LIN {X 0,Y 418.246,Z 332.012,A -85,B 0,C 180,E1 -10220.619,E2 -10220.619} C_VEL
LIN {X 0,Y 418.235,Z 332.015,A -85,B 0,C 180,E1 -10223.975,E2 -10223.975} C_VEL
LIN {X 0,Y 418.248,Z 332.008,A -85,B 0,C 180,E1 -10227.156,E2 -10227.156} C_VEL
LIN {X 0,Y 418.251,Z 331.996,A -85,B 0,C 180,E1 -10230.837,E2 -10230.837} C_VEL
LIN {X 0,Y 418.226,Z 332.013,A -85,B 0,C 180,E1 -10234.093,E2 -10234.093} C_VEL
LIN {X 0,Y 418.221,Z 332.012,A -85,B 0,C 180,E1 -10237.263,E2 -10237.263} C_VEL
LIN {X 0,Y 418.272,Z 332.006,A -85,B 0,C 180,E1 -10240.364,E2 -10240.364} C_VEL
LIN {X 0,Y 418.304,Z 332.002,A -85,B 0,C 180,E1 -10243.404,E2 -10243.404} C_VEL
LIN {X 0,Y 418.334,Z 331.998,A -85,B 0,C 180,E1 -10247,E2 -10247} C_VEL
LIN {X 0,Y 418.306,Z 332.002,A -85,B 0,C 180,E1 -10250.328,E2 -10250.328} C_VEL
LIN {X 0,Y 418.43,Z 331.983,A -85,B 0,C 180,E1 -10253.248,E2 -10253.248} C_VEL
LIN {X 0,Y 418.304,Z 332.004,A -85,B 0,C 180,E1 -10255.181,E2 -10255.181} C_VEL
LIN {X 0,Y 418.521,Z 331.97,A -85,B 0,C 180,E1 -10258.076,E2 -10258.076} C_VEL
LIN {X 0,Y 418.395,Z 331.993,A -85,B 0,C 180,E1 -10260.963,E2 -10260.963} C_VEL
LIN {X 0,Y 418.478,Z 331.976,A -85,B 0,C 180,E1 -10262.888,E2 -10262.888} C_VEL
LIN {X 0,Y 418.453,Z 331.982,A -85,B 0,C 180,E1 -10266.598,E2 -10266.598} C_VEL
LIN {X 0,Y 418.325,Z 332.001,A -85,B 0,C 180,E1 -10269.672,E2 -10269.672} C_VEL
LIN {X 0,Y 418.336,Z 331.996,A -85,B 0,C 180,E1 -10273.001,E2 -10273.001} C_VEL
LIN {X 0,Y 418.302,Z 332,A -85,B 0,C 180,E1 -10276.736,E2 -10276.736} C_VEL
LIN {X 0,Y 418.261,Z 332.005,A -85,B 0,C 180,E1 -10279.791,E2 -10279.791} C_VEL
LIN {X 0,Y 418.224,Z 332.016,A -85,B 0,C 180,E1 -10282.737,E2 -10282.737} C_VEL
LIN {X 0,Y 418.263,Z 332.006,A -85,B 0,C 180,E1 -10285.905,E2 -10285.905} C_VEL
LIN {X 0,Y 418.258,Z 332.01,A -85,B 0,C 180,E1 -10289.163,E2 -10289.163} C_VEL
LIN {X 0,Y 418.251,Z 332.012,A -85,B 0,C 180,E1 -10292.845,E2 -10292.845} C_VEL
LIN {X 0,Y 418.239,Z 332.012,A -85,B 0,C 180,E1 -10296.239,E2 -10296.239} C_VEL
LIN {X 0,Y 418.24,Z 332.008,A -85,B 0,C 180,E1 -10299.684,E2 -10299.684} C_VEL
LIN {X 0,Y 418.226,Z 332.014,A -85,B 0,C 180,E1 -10302.322,E2 -10302.322} C_VEL
LIN {X 0,Y 418.233,Z 332.013,A -85,B 0,C 180,E1 -10305.11,E2 -10305.11} C_VEL
LIN {X 0,Y 418.238,Z 332.013,A -85,B 0,C 180,E1 -10307.768,E2 -10307.768} C_VEL
LIN {X 0,Y 418.259,Z 332.011,A -85,B 0,C 180,E1 -10310.619,E2 -10310.619} C_VEL
LIN {X 0,Y 418.246,Z 332.014,A -85,B 0,C 180,E1 -10313.977,E2 -10313.977} C_VEL
LIN {X 0,Y 418.258,Z 332.108,A -85,B 0,C 180,E1 -10317.157,E2 -10317.157} C_VEL
LIN {X 0,Y 421.168,Z 344.799,A -85,B 0,C 180,E1 -10320.196,E2 -10320.196} C_VEL
LIN {X 0,Y 421.536,Z 346.615,A -85,B 0,C 180,E1 -10320.615,E2 -10320.615} C_VEL
LIN {X 0,Y 424.436,Z 354.758,A -85,B 0,C 180,E1 -10320.961,E2 -10320.961} C_VEL
LIN {X 0,Y 427.981,Z 370.411,A -85,B 0,C 180,E1 -10321.469,E2 -10321.469} C_VEL
LIN {X 0,Y 426.182,Z 483.541,A -85,B 0,C 180,E1 -10323.429,E2 -10323.429} C_VEL
LIN {X 0,Y 425.633,Z 498.284,A -85,B 0,C 180,E1 -10323.888,E2 -10323.888} C_VEL
LIN {X 0,Y 424.959,Z 512.346,A -85,B 0,C 180,E1 -10324.534,E2 -10324.534} C_VEL
LIN {X 0,Y 424.111,Z 524.49,A -85,B 0,C 180,E1 -10325.266,E2 -10325.266} C_VEL
LIN {X 0,Y 423.088,Z 537.105,A -85,B 0,C 180,E1 -10326.23,E2 -10326.23} C_VEL
LIN {X 0,Y 422.044,Z 548.902,A -85,B 0,C 180,E1 -10327.352,E2 -10327.352} C_VEL
LIN {X 0,Y 421.019,Z 559.619,A -85,B 0,C 180,E1 -10328.596,E2 -10328.596} C_VEL
LIN {X 0,Y 420.156,Z 569.213,A -85,B 0,C 180,E1 -10329.947,E2 -10329.947} C_VEL
LIN {X 0,Y 419.256,Z 577.982,A -85,B 0,C 180,E1 -10331.428,E2 -10331.428} C_VEL
LIN {X 0,Y 418.484,Z 586.467,A -85,B 0,C 180,E1 -10333.189,E2 -10333.189} C_VEL
LIN {X 0,Y 417.905,Z 593.022,A -85,B 0,C 180,E1 -10334.891,E2 -10334.891} C_VEL
LIN {X 0,Y 417.698,Z 595.505,A -85,B 0,C 180,E1 -10335.661,E2 -10335.661} C_VEL
LIN {X 0,Y 416.879,Z 597.766,A -85,B 0,C 180,E1 -10336.404,E2 -10336.404} C_VEL
LIN {X 0,Y 413.8,Z 601.016,A -85,B 0,C 180,E1 -10337.624,E2 -10337.624} C_VEL
LIN {X 0,Y 411.23,Z 603.194,A -85,B 0,C 180,E1 -10338.629,E2 -10338.629} C_VEL
LIN {X 0,Y 410.083,Z 604.573,A -85,B 0,C 180,E1 -10339.42,E2 -10339.42} C_VEL
LIN {X 0,Y 409.964,Z 604.953,A -85,B 0,C 180,E1 -10339.69,E2 -10339.69} C_VEL
LIN {X 0,Y 409.89,Z 606.657,A -85,B 0,C 180,E1 -10341.123,E2 -10341.123} C_VEL
LIN {X 0,Y 409.943,Z 607.798,A -85,B 0,C 180,E1 -10343.108,E2 -10343.108} C_VEL
LIN {X 0,Y 409.98,Z 607.87,A -85,B 0,C 180,E1 -10344.097,E2 -10344.097} C_VEL
LIN {X 0,Y 409.924,Z 607.031,A -85,B 0,C 180,E1 -10346.068,E2 -10346.068} C_VEL
LIN {X 0,Y 410.03,Z 604.86,A -85,B 0,C 180,E1 -10348.036,E2 -10348.036} C_VEL
LIN {X 0,Y 410.104,Z 601.318,A -85,B 0,C 180,E1 -10350,E2 -10350} C_VEL
LIN {X 0,Y 410.342,Z 596.299,A -85,B 0,C 180,E1 -10351.963,E2 -10351.963} C_VEL
LIN {X 0,Y 410.74,Z 591.435,A -85,B 0,C 180,E1 -10353.433,E2 -10353.433} C_VEL
LIN {X 0,Y 411.265,Z 584.464,A -85,B 0,C 180,E1 -10355.147,E2 -10355.147} C_VEL
LIN {X 0,Y 412.002,Z 577.174,A -85,B 0,C 180,E1 -10356.612,E2 -10356.612} C_VEL
LIN {X 0,Y 412.81,Z 568.431,A -85,B 0,C 180,E1 -10358.074,E2 -10358.074} C_VEL
LIN {X 0,Y 413.732,Z 557.988,A -85,B 0,C 180,E1 -10359.516,E2 -10359.516} C_VEL
LIN {X 0,Y 414.646,Z 547.174,A -85,B 0,C 180,E1 -10360.745,E2 -10360.745} C_VEL
LIN {X 0,Y 415.586,Z 535.499,A -85,B 0,C 180,E1 -10361.832,E2 -10361.832} C_VEL
LIN {X 0,Y 416.513,Z 522.632,A -85,B 0,C 180,E1 -10362.795,E2 -10362.795} C_VEL
LIN {X 0,Y 417.36,Z 509.181,A -85,B 0,C 180,E1 -10363.573,E2 -10363.573} C_VEL
LIN {X 0,Y 417.958,Z 495.939,A -85,B 0,C 180,E1 -10364.143,E2 -10364.143} C_VEL
LIN {X 0,Y 418.392,Z 481.346,A -85,B 0,C 180,E1 -10364.562,E2 -10364.562} C_VEL
LIN {X 0,Y 419.816,Z 370.702,A -85,B 0,C 180,E1 -10366.485,E2 -10366.485} C_VEL
LIN {X 0,Y 415.593,Z 351.069,A -85,B 0,C 180,E1 -10367.062,E2 -10367.062} C_VEL
LIN {X 0,Y 414.048,Z 346.577,A -85,B 0,C 180,E1 -10367.248,E2 -10367.248} C_VEL
LIN {X 0,Y 411.854,Z 335.866,A -85,B 0,C 180,E1 -10369.695,E2 -10369.695} C_VEL
LIN {X 0,Y 411.239,Z 332.889,A -85,B 0,C 180,E1 -10370.435,E2 -10370.435} C_VEL
LIN {X 0,Y 411.228,Z 332.887,A -85,B 0,C 180,E1 -10374.215,E2 -10374.215} C_VEL
LIN {X 0,Y 411.261,Z 332.883,A -85,B 0,C 180,E1 -10377.477,E2 -10377.477} C_VEL
LIN {X 0,Y 411.19,Z 332.888,A -85,B 0,C 180,E1 -10380.847,E2 -10380.847} C_VEL
LIN {X 0,Y 411.206,Z 332.885,A -85,B 0,C 180,E1 -10384.332,E2 -10384.332} C_VEL
LIN {X 0,Y 411.199,Z 332.889,A -85,B 0,C 180,E1 -10387.972,E2 -10387.972} C_VEL
LIN {X 0,Y 411.18,Z 332.876,A -85,B 0,C 180,E1 -10390.503,E2 -10390.503} C_VEL
LIN {X 0,Y 411.171,Z 332.892,A -85,B 0,C 180,E1 -10393.132,E2 -10393.132} C_VEL
LIN {X 0,Y 411.164,Z 332.893,A -85,B 0,C 180,E1 -10395.88,E2 -10395.88} C_VEL
LIN {X 0,Y 411.159,Z 332.888,A -85,B 0,C 180,E1 -10398.771,E2 -10398.771} C_VEL
LIN {X 0,Y 411.186,Z 332.883,A -85,B 0,C 180,E1 -10402.025,E2 -10402.025} C_VEL
LIN {X 0,Y 411.198,Z 332.885,A -85,B 0,C 180,E1 -10405.665,E2 -10405.665} C_VEL
LIN {X 0,Y 411.182,Z 332.895,A -85,B 0,C 180,E1 -10409.151,E2 -10409.151} C_VEL
LIN {X 0,Y 411.251,Z 332.872,A -85,B 0,C 180,E1 -10412.521,E2 -10412.521} C_VEL
LIN {X 0,Y 411.202,Z 332.886,A -85,B 0,C 180,E1 -10415.783,E2 -10415.783} C_VEL
LIN {X 0,Y 411.186,Z 332.88,A -85,B 0,C 180,E1 -10418.965,E2 -10418.965} C_VEL
LIN {X 0,Y 411.235,Z 332.879,A -85,B 0,C 180,E1 -10422.084,E2 -10422.084} C_VEL
LIN {X 0,Y 411.247,Z 332.878,A -85,B 0,C 180,E1 -10425.146,E2 -10425.146} C_VEL
LIN {X 0,Y 411.27,Z 332.866,A -85,B 0,C 180,E1 -10428.166,E2 -10428.166} C_VEL
LIN {X 0,Y 411.427,Z 332.859,A -85,B 0,C 180,E1 -10432.191,E2 -10432.191} C_VEL
LIN {X 0,Y 411.432,Z 332.853,A -85,B 0,C 180,E1 -10434.117,E2 -10434.117} C_VEL
LIN {X 0,Y 411.493,Z 332.847,A -85,B 0,C 180,E1 -10438.042,E2 -10438.042} C_VEL
LIN {X 0,Y 411.487,Z 332.848,A -85,B 0,C 180,E1 -10441.957,E2 -10441.957} C_VEL
LIN {X 0,Y 411.405,Z 332.861,A -85,B 0,C 180,E1 -10445.883,E2 -10445.883} C_VEL
LIN {X 0,Y 411.298,Z 332.867,A -85,B 0,C 180,E1 -10448.846,E2 -10448.846} C_VEL
LIN {X 0,Y 411.269,Z 332.878,A -85,B 0,C 180,E1 -10451.833,E2 -10451.833} C_VEL
LIN {X 0,Y 411.247,Z 332.875,A -85,B 0,C 180,E1 -10454.853,E2 -10454.853} C_VEL
LIN {X 0,Y 411.233,Z 332.883,A -85,B 0,C 180,E1 -10457.916,E2 -10457.916} C_VEL
LIN {X 0,Y 411.185,Z 332.879,A -85,B 0,C 180,E1 -10461.034,E2 -10461.034} C_VEL
LIN {X 0,Y 411.201,Z 332.888,A -85,B 0,C 180,E1 -10464.217,E2 -10464.217} C_VEL
LIN {X 0,Y 411.179,Z 332.887,A -85,B 0,C 180,E1 -10467.483,E2 -10467.483} C_VEL
LIN {X 0,Y 411.179,Z 332.886,A -85,B 0,C 180,E1 -10470.848,E2 -10470.848} C_VEL
LIN {X 0,Y 411.197,Z 332.888,A -85,B 0,C 180,E1 -10474.334,E2 -10474.334} C_VEL
LIN {X 0,Y 411.188,Z 332.892,A -85,B 0,C 180,E1 -10477.974,E2 -10477.974} C_VEL
LIN {X 0,Y 411.175,Z 332.884,A -85,B 0,C 180,E1 -10480.505,E2 -10480.505} C_VEL
LIN {X 0,Y 411.167,Z 332.889,A -85,B 0,C 180,E1 -10483.134,E2 -10483.134} C_VEL
LIN {X 0,Y 411.162,Z 332.896,A -85,B 0,C 180,E1 -10485.882,E2 -10485.882} C_VEL
LIN {X 0,Y 411.157,Z 332.893,A -85,B 0,C 180,E1 -10488.773,E2 -10488.773} C_VEL
LIN {X 0,Y 411.187,Z 332.895,A -85,B 0,C 180,E1 -10492.027,E2 -10492.027} C_VEL
LIN {X 0,Y 411.203,Z 332.894,A -85,B 0,C 180,E1 -10495.667,E2 -10495.667} C_VEL
LIN {X 0,Y 411.188,Z 332.893,A -85,B 0,C 180,E1 -10499.153,E2 -10499.153} C_VEL
LIN {X 0,Y 411.232,Z 332.987,A -85,B 0,C 180,E1 -10500.044,E2 -10500.044} C_VEL
LIN {X 0,Y 414.112,Z 345.944,A -85,B 0,C 180,E1 -10502.728,E2 -10502.728} C_VEL
LIN {X 0,Y 415.486,Z 353.214,A -85,B 0,C 180,E1 -10504.18,E2 -10504.18} C_VEL
LIN {X 0,Y 414.529,Z 367.772,A -85,B 0,C 180,E1 -10506.824,E2 -10506.824} C_VEL
LIN {X 0,Y 419.611,Z 397.438,A -85,B 0,C 180,E1 -10507.622,E2 -10507.622} C_VEL
LIN {X 0,Y 418.121,Z 505.146,A -85,B 0,C 180,E1 -10509.492,E2 -10509.492} C_VEL
LIN {X 0,Y 417.563,Z 519.304,A -85,B 0,C 180,E1 -10509.913,E2 -10509.913} C_VEL
LIN {X 0,Y 416.82,Z 532.559,A -85,B 0,C 180,E1 -10510.49,E2 -10510.49} C_VEL
LIN {X 0,Y 416.007,Z 545.949,A -85,B 0,C 180,E1 -10511.278,E2 -10511.278} C_VEL
LIN {X 0,Y 415.023,Z 558.885,A -85,B 0,C 180,E1 -10512.254,E2 -10512.254} C_VEL
LIN {X 0,Y 413.918,Z 570.625,A -85,B 0,C 180,E1 -10513.351,E2 -10513.351} C_VEL
LIN {X 0,Y 413.086,Z 580.397,A -85,B 0,C 180,E1 -10514.458,E2 -10514.458} C_VEL
LIN {X 0,Y 412.209,Z 591.218,A -85,B 0,C 180,E1 -10515.939,E2 -10515.939} C_VEL
LIN {X 0,Y 411.522,Z 600.144,A -85,B 0,C 180,E1 -10517.424,E2 -10517.424} C_VEL
LIN {X 0,Y 410.96,Z 607.561,A -85,B 0,C 180,E1 -10518.908,E2 -10518.908} C_VEL
LIN {X 0,Y 410.45,Z 614.649,A -85,B 0,C 180,E1 -10520.639,E2 -10520.639} C_VEL
LIN {X 0,Y 410.157,Z 621.011,A -85,B 0,C 180,E1 -10522.617,E2 -10522.617} C_VEL
LIN {X 0,Y 410.034,Z 624.648,A -85,B 0,C 180,E1 -10524.097,E2 -10524.097} C_VEL
LIN {X 0,Y 409.92,Z 628.205,A -85,B 0,C 180,E1 -10526.068,E2 -10526.068} C_VEL
LIN {X 0,Y 409.964,Z 630.356,A -85,B 0,C 180,E1 -10528.035,E2 -10528.035} C_VEL
LIN {X 0,Y 409.924,Z 631.15,A -85,B 0,C 180,E1 -10530,E2 -10530} C_VEL
LIN {X 0,Y 409.964,Z 630.613,A -85,B 0,C 180,E1 -10531.965,E2 -10531.965} C_VEL
LIN {X 0,Y 409.919,Z 628.737,A -85,B 0,C 180,E1 -10533.932,E2 -10533.932} C_VEL
LIN {X 0,Y 410.034,Z 625.471,A -85,B 0,C 180,E1 -10535.903,E2 -10535.903} C_VEL
LIN {X 0,Y 410.161,Z 622.032,A -85,B 0,C 180,E1 -10537.383,E2 -10537.383} C_VEL
LIN {X 0,Y 410.51,Z 616.109,A -85,B 0,C 180,E1 -10539.36,E2 -10539.36} C_VEL
LIN {X 0,Y 411.005,Z 609.456,A -85,B 0,C 180,E1 -10541.091,E2 -10541.091} C_VEL
LIN {X 0,Y 411.737,Z 601.197,A -85,B 0,C 180,E1 -10542.82,E2 -10542.82} C_VEL
LIN {X 0,Y 412.532,Z 592.598,A -85,B 0,C 180,E1 -10544.301,E2 -10544.301} C_VEL
LIN {X 0,Y 413.546,Z 582.197,A -85,B 0,C 180,E1 -10545.778,E2 -10545.778} C_VEL
LIN {X 0,Y 414.765,Z 570.585,A -85,B 0,C 180,E1 -10547.122,E2 -10547.122} C_VEL
LIN {X 0,Y 415.872,Z 559.001,A -85,B 0,C 180,E1 -10548.218,E2 -10548.218} C_VEL
LIN {X 0,Y 416.962,Z 546.906,A -85,B 0,C 180,E1 -10549.142,E2 -10549.142} C_VEL
LIN {X 0,Y 417.909,Z 533.112,A -85,B 0,C 180,E1 -10549.974,E2 -10549.974} C_VEL
LIN {X 0,Y 418.786,Z 519.614,A -85,B 0,C 180,E1 -10550.571,E2 -10550.571} C_VEL
LIN {X 0,Y 419.409,Z 505.937,A -85,B 0,C 180,E1 -10550.988,E2 -10550.988} C_VEL
LIN {X 0,Y 421.196,Z 399.896,A -85,B 0,C 180,E1 -10552.852,E2 -10552.852} C_VEL
LIN {X 0,Y 420.511,Z 393.745,A -85,B 0,C 180,E1 -10553.008,E2 -10553.008} C_VEL
LIN {X 0,Y 415.325,Z 367.391,A -85,B 0,C 180,E1 -10553.851,E2 -10553.851} C_VEL
LIN {X 0,Y 416.283,Z 355.716,A -85,B 0,C 180,E1 -10556.036,E2 -10556.036} C_VEL
LIN {X 0,Y 414.111,Z 344.618,A -85,B 0,C 180,E1 -10558.371,E2 -10558.371} C_VEL
LIN {X 0,Y 411.208,Z 332.891,A -85,B 0,C 180,E1 -10561.008,E2 -10561.008} C_VEL
LIN {X 0,Y 411.202,Z 332.891,A -85,B 0,C 180,E1 -10564.333,E2 -10564.333} C_VEL
LIN {X 0,Y 411.19,Z 332.882,A -85,B 0,C 180,E1 -10567.973,E2 -10567.973} C_VEL
LIN {X 0,Y 411.158,Z 332.886,A -85,B 0,C 180,E1 -10571.227,E2 -10571.227} C_VEL
LIN {X 0,Y 411.169,Z 332.889,A -85,B 0,C 180,E1 -10574.49,E2 -10574.49} C_VEL
LIN {X 0,Y 411.17,Z 332.893,A -85,B 0,C 180,E1 -10578.194,E2 -10578.194} C_VEL
LIN {X 0,Y 411.21,Z 332.887,A -85,B 0,C 180,E1 -10580.775,E2 -10580.775} C_VEL
LIN {X 0,Y 411.19,Z 332.888,A -85,B 0,C 180,E1 -10584.471,E2 -10584.471} C_VEL
LIN {X 0,Y 411.199,Z 332.887,A -85,B 0,C 180,E1 -10586.873,E2 -10586.873} C_VEL
LIN {X 0,Y 411.203,Z 332.872,A -85,B 0,C 180,E1 -10590.649,E2 -10590.649} C_VEL
LIN {X 0,Y 411.185,Z 332.891,A -85,B 0,C 180,E1 -10593.616,E2 -10593.616} C_VEL
LIN {X 0,Y 411.185,Z 332.888,A -85,B 0,C 180,E1 -10596.852,E2 -10596.852} C_VEL
LIN {X 0,Y 411.203,Z 332.887,A -85,B 0,C 180,E1 -10600.051,E2 -10600.051} C_VEL
LIN {X 0,Y 411.252,Z 332.88,A -85,B 0,C 180,E1 -10603.131,E2 -10603.131} C_VEL
LIN {X 0,Y 411.293,Z 332.875,A -85,B 0,C 180,E1 -10606.897,E2 -10606.897} C_VEL
LIN {X 0,Y 411.26,Z 332.88,A -85,B 0,C 180,E1 -10610.161,E2 -10610.161} C_VEL
LIN {X 0,Y 411.379,Z 332.861,A -85,B 0,C 180,E1 -10613.132,E2 -10613.132} C_VEL
LIN {X 0,Y 411.276,Z 332.879,A -85,B 0,C 180,E1 -10615.099,E2 -10615.099} C_VEL
LIN {X 0,Y 411.49,Z 332.846,A -85,B 0,C 180,E1 -10618.043,E2 -10618.043} C_VEL
LIN {X 0,Y 411.497,Z 332.845,A -85,B 0,C 180,E1 -10621.958,E2 -10621.958} C_VEL
LIN {X 0,Y 411.412,Z 332.859,A -85,B 0,C 180,E1 -10626.6,E2 -10626.6} C_VEL
LIN {X 0,Y 411.307,Z 332.872,A -85,B 0,C 180,E1 -10628.847,E2 -10628.847} C_VEL
LIN {X 0,Y 411.27,Z 332.871,A -85,B 0,C 180,E1 -10631.834,E2 -10631.834} C_VEL
LIN {X 0,Y 411.247,Z 332.885,A -85,B 0,C 180,E1 -10634.854,E2 -10634.854} C_VEL
LIN {X 0,Y 411.236,Z 332.882,A -85,B 0,C 180,E1 -10637.916,E2 -10637.916} C_VEL
LIN {X 0,Y 411.187,Z 332.888,A -85,B 0,C 180,E1 -10641.035,E2 -10641.035} C_VEL
LIN {X 0,Y 411.212,Z 332.884,A -85,B 0,C 180,E1 -10644.217,E2 -10644.217} C_VEL
LIN {X 0,Y 411.252,Z 332.878,A -85,B 0,C 180,E1 -10647.479,E2 -10647.479} C_VEL
LIN {X 0,Y 411.183,Z 332.889,A -85,B 0,C 180,E1 -10650.849,E2 -10650.849} C_VEL
LIN {X 0,Y 411.2,Z 332.887,A -85,B 0,C 180,E1 -10654.335,E2 -10654.335} C_VEL
LIN {X 0,Y 411.186,Z 332.886,A -85,B 0,C 180,E1 -10657.975,E2 -10657.975} C_VEL
LIN {X 0,Y 411.159,Z 332.893,A -85,B 0,C 180,E1 -10661.229,E2 -10661.229} C_VEL
LIN {X 0,Y 411.173,Z 332.893,A -85,B 0,C 180,E1 -10664.492,E2 -10664.492} C_VEL
LIN {X 0,Y 411.175,Z 332.895,A -85,B 0,C 180,E1 -10668.196,E2 -10668.196} C_VEL
LIN {X 0,Y 411.223,Z 332.888,A -85,B 0,C 180,E1 -10670.778,E2 -10670.778} C_VEL
LIN {X 0,Y 411.199,Z 332.887,A -85,B 0,C 180,E1 -10674.473,E2 -10674.473} C_VEL
LIN {X 0,Y 411.227,Z 333.001,A -85,B 0,C 180,E1 -10676.774,E2 -10676.774} C_VEL
LIN {X 0,Y 414.352,Z 346.613,A -85,B 0,C 180,E1 -10680.095,E2 -10680.095} C_VEL
LIN {X 0,Y 414.484,Z 347.202,A -85,B 0,C 180,E1 -10680.167,E2 -10680.167} C_VEL
LIN {X 0,Y 418.19,Z 356.786,A -85,B 0,C 180,E1 -10680.595,E2 -10680.595} C_VEL
LIN {X 0,Y 421.558,Z 371.616,A -85,B 0,C 180,E1 -10681.088,E2 -10681.088} C_VEL
LIN {X 0,Y 419.636,Z 483.745,A -85,B 0,C 180,E1 -10683.058,E2 -10683.058} C_VEL
LIN {X 0,Y 419.091,Z 498.27,A -85,B 0,C 180,E1 -10683.516,E2 -10683.516} C_VEL
LIN {X 0,Y 418.362,Z 512.383,A -85,B 0,C 180,E1 -10684.17,E2 -10684.17} C_VEL
LIN {X 0,Y 417.409,Z 525.458,A -85,B 0,C 180,E1 -10684.974,E2 -10684.974} C_VEL
LIN {X 0,Y 416.369,Z 537.689,A -85,B 0,C 180,E1 -10685.933,E2 -10685.933} C_VEL
LIN {X 0,Y 415.361,Z 548.417,A -85,B 0,C 180,E1 -10686.967,E2 -10686.967} C_VEL
LIN {X 0,Y 414.346,Z 558.16,A -85,B 0,C 180,E1 -10688.09,E2 -10688.09} C_VEL
LIN {X 0,Y 413.431,Z 568.078,A -85,B 0,C 180,E1 -10689.47,E2 -10689.47} C_VEL
LIN {X 0,Y 412.376,Z 577.785,A -85,B 0,C 180,E1 -10691.107,E2 -10691.107} C_VEL
LIN {X 0,Y 411.689,Z 585.113,A -85,B 0,C 180,E1 -10692.619,E2 -10692.619} C_VEL
LIN {X 0,Y 411.096,Z 591.175,A -85,B 0,C 180,E1 -10694.126,E2 -10694.126} C_VEL
LIN {X 0,Y 410.647,Z 596.17,A -85,B 0,C 180,E1 -10695.632,E2 -10695.632} C_VEL
LIN {X 0,Y 410.302,Z 601.035,A -85,B 0,C 180,E1 -10697.516,E2 -10697.516} C_VEL
LIN {X 0,Y 410.06,Z 604.154,A -85,B 0,C 180,E1 -10699.133,E2 -10699.133} C_VEL
LIN {X 0,Y 409.964,Z 604.953,A -85,B 0,C 180,E1 -10699.69,E2 -10699.69} C_VEL
LIN {X 0,Y 409.241,Z 606.048,A -85,B 0,C 180,E1 -10700.496,E2 -10700.496} C_VEL
LIN {X 0,Y 406.418,Z 607.421,A -85,B 0,C 180,E1 -10701.816,E2 -10701.816} C_VEL
LIN {X 0,Y 404.05,Z 608.026,A -85,B 0,C 180,E1 -10702.889,E2 -10702.889} C_VEL
LIN {X 0,Y 403.004,Z 608.126,A -85,B 0,C 180,E1 -10703.719,E2 -10703.719} C_VEL
LIN {X 0,Y 402.901,Z 608.082,A -85,B 0,C 180,E1 -10704,E2 -10704} C_VEL
LIN {X 0,Y 402.84,Z 607.29,A -85,B 0,C 180,E1 -10705.998,E2 -10705.998} C_VEL
LIN {X 0,Y 402.957,Z 605.165,A -85,B 0,C 180,E1 -10708.001,E2 -10708.001} C_VEL
LIN {X 0,Y 403.019,Z 601.673,A -85,B 0,C 180,E1 -10710,E2 -10710} C_VEL
LIN {X 0,Y 403.262,Z 596.705,A -85,B 0,C 180,E1 -10711.997,E2 -10711.997} C_VEL
LIN {X 0,Y 403.752,Z 590.109,A -85,B 0,C 180,E1 -10713.992,E2 -10713.992} C_VEL
LIN {X 0,Y 404.512,Z 582.752,A -85,B 0,C 180,E1 -10715.733,E2 -10715.733} C_VEL
LIN {X 0,Y 405.267,Z 575.079,A -85,B 0,C 180,E1 -10717.223,E2 -10717.223} C_VEL
LIN {X 0,Y 406.132,Z 565.865,A -85,B 0,C 180,E1 -10718.709,E2 -10718.709} C_VEL
LIN {X 0,Y 407.011,Z 555.701,A -85,B 0,C 180,E1 -10720.067,E2 -10720.067} C_VEL
LIN {X 0,Y 408.003,Z 544.479,A -85,B 0,C 180,E1 -10721.299,E2 -10721.299} C_VEL
LIN {X 0,Y 409.005,Z 532.093,A -85,B 0,C 180,E1 -10722.403,E2 -10722.403} C_VEL
LIN {X 0,Y 409.894,Z 520.134,A -85,B 0,C 180,E1 -10723.257,E2 -10723.257} C_VEL
LIN {X 0,Y 410.686,Z 507.015,A -85,B 0,C 180,E1 -10723.988,E2 -10723.988} C_VEL
LIN {X 0,Y 411.368,Z 493.66,A -85,B 0,C 180,E1 -10724.532,E2 -10724.532} C_VEL
LIN {X 0,Y 411.735,Z 478.975,A -85,B 0,C 180,E1 -10724.93,E2 -10724.93} C_VEL
LIN {X 0,Y 413.261,Z 372.068,A -85,B 0,C 180,E1 -10726.804,E2 -10726.804} C_VEL
LIN {X 0,Y 409.161,Z 353.235,A -85,B 0,C 180,E1 -10727.372,E2 -10727.372} C_VEL
LIN {X 0,Y 406.897,Z 346.78,A -85,B 0,C 180,E1 -10727.641,E2 -10727.641} C_VEL
LIN {X 0,Y 404.186,Z 333.781,A -85,B 0,C 180,E1 -10730.682,E2 -10730.682} C_VEL
LIN {X 0,Y 404.171,Z 333.767,A -85,B 0,C 180,E1 -10733.574,E2 -10733.574} C_VEL
LIN {X 0,Y 404.185,Z 333.766,A -85,B 0,C 180,E1 -10735.765,E2 -10735.765} C_VEL
LIN {X 0,Y 404.197,Z 333.76,A -85,B 0,C 180,E1 -10737.999,E2 -10737.999} C_VEL
LIN {X 0,Y 404.14,Z 333.77,A -85,B 0,C 180,E1 -10741.557,E2 -10741.557} C_VEL
LIN {X 0,Y 404.185,Z 333.76,A -85,B 0,C 180,E1 -10745.015,E2 -10745.015} C_VEL
LIN {X 0,Y 404.157,Z 333.764,A -85,B 0,C 180,E1 -10748.755,E2 -10748.755} C_VEL
LIN {X 0,Y 404.121,Z 333.765,A -85,B 0,C 180,E1 -10751.598,E2 -10751.598} C_VEL
LIN {X 0,Y 404.142,Z 333.763,A -85,B 0,C 180,E1 -10754.521,E2 -10754.521} C_VEL
LIN {X 0,Y 404.132,Z 333.771,A -85,B 0,C 180,E1 -10757.294,E2 -10757.294} C_VEL
LIN {X 0,Y 404.165,Z 333.764,A -85,B 0,C 180,E1 -10759.954,E2 -10759.954} C_VEL
LIN {X 0,Y 404.13,Z 333.767,A -85,B 0,C 180,E1 -10763.124,E2 -10763.124} C_VEL
LIN {X 0,Y 404.138,Z 333.762,A -85,B 0,C 180,E1 -10766.186,E2 -10766.186} C_VEL
LIN {X 0,Y 404.138,Z 333.766,A -85,B 0,C 180,E1 -10769.714,E2 -10769.714} C_VEL
LIN {X 0,Y 404.185,Z 333.754,A -85,B 0,C 180,E1 -10773.122,E2 -10773.122} C_VEL
LIN {X 0,Y 404.151,Z 333.765,A -85,B 0,C 180,E1 -10776.424,E2 -10776.424} C_VEL
LIN {X 0,Y 404.182,Z 333.747,A -85,B 0,C 180,E1 -10779.873,E2 -10779.873} C_VEL
LIN {X 0,Y 404.206,Z 333.763,A -85,B 0,C 180,E1 -10782.992,E2 -10782.992} C_VEL
LIN {X 0,Y 404.273,Z 333.738,A -85,B 0,C 180,E1 -10786.938,E2 -10786.938} C_VEL
LIN {X 0,Y 404.243,Z 333.75,A -85,B 0,C 180,E1 -10789.988,E2 -10789.988} C_VEL
LIN {X 0,Y 404.371,Z 333.735,A -85,B 0,C 180,E1 -10793.012,E2 -10793.012} C_VEL
LIN {X 0,Y 404.257,Z 333.737,A -85,B 0,C 180,E1 -10795.013,E2 -10795.013} C_VEL
LIN {X 0,Y 404.462,Z 333.722,A -85,B 0,C 180,E1 -10798.008,E2 -10798.008} C_VEL
LIN {X 0,Y 404.456,Z 333.724,A -85,B 0,C 180,E1 -10801.991,E2 -10801.991} C_VEL
LIN {X 0,Y 404.355,Z 333.74,A -85,B 0,C 180,E1 -10805.986,E2 -10805.986} C_VEL
LIN {X 0,Y 404.247,Z 333.744,A -85,B 0,C 180,E1 -10809.002,E2 -10809.002} C_VEL
LIN {X 0,Y 404.242,Z 333.755,A -85,B 0,C 180,E1 -10812.042,E2 -10812.042} C_VEL
LIN {X 0,Y 404.193,Z 333.752,A -85,B 0,C 180,E1 -10815.118,E2 -10815.118} C_VEL
LIN {X 0,Y 404.192,Z 333.764,A -85,B 0,C 180,E1 -10818.239,E2 -10818.239} C_VEL
LIN {X 0,Y 404.127,Z 333.758,A -85,B 0,C 180,E1 -10821.42,E2 -10821.42} C_VEL
LIN {X 0,Y 404.154,Z 333.762,A -85,B 0,C 180,E1 -10824.667,E2 -10824.667} C_VEL
LIN {X 0,Y 404.12,Z 333.772,A -85,B 0,C 180,E1 -10828.005,E2 -10828.005} C_VEL
LIN {X 0,Y 404.135,Z 333.765,A -85,B 0,C 180,E1 -10830.286,E2 -10830.286} C_VEL
LIN {X 0,Y 404.136,Z 333.768,A -85,B 0,C 180,E1 -10833.813,E2 -10833.813} C_VEL
LIN {X 0,Y 404.128,Z 333.766,A -85,B 0,C 180,E1 -10836.876,E2 -10836.876} C_VEL
LIN {X 0,Y 404.14,Z 333.764,A -85,B 0,C 180,E1 -10840.081,E2 -10840.081} C_VEL
LIN {X 0,Y 404.146,Z 333.764,A -85,B 0,C 180,E1 -10843.084,E2 -10843.084} C_VEL
LIN {X 0,Y 404.142,Z 333.77,A -85,B 0,C 180,E1 -10845.927,E2 -10845.927} C_VEL
LIN {X 0,Y 404.112,Z 333.77,A -85,B 0,C 180,E1 -10848.636,E2 -10848.636} C_VEL
LIN {X 0,Y 404.145,Z 333.773,A -85,B 0,C 180,E1 -10851.494,E2 -10851.494} C_VEL
LIN {X 0,Y 404.181,Z 333.768,A -85,B 0,C 180,E1 -10854.985,E2 -10854.985} C_VEL
LIN {X 0,Y 404.139,Z 333.77,A -85,B 0,C 180,E1 -10858.555,E2 -10858.555} C_VEL
LIN {X 0,Y 404.17,Z 333.819,A -85,B 0,C 180,E1 -10859.718,E2 -10859.718} C_VEL
LIN {X 0,Y 407.113,Z 346.963,A -85,B 0,C 180,E1 -10862.498,E2 -10862.498} C_VEL
LIN {X 0,Y 408.573,Z 354.383,A -85,B 0,C 180,E1 -10864.012,E2 -10864.012} C_VEL
LIN {X 0,Y 407.668,Z 367.447,A -85,B 0,C 180,E1 -10866.444,E2 -10866.444} C_VEL
LIN {X 0,Y 412.999,Z 398.828,A -85,B 0,C 180,E1 -10867.309,E2 -10867.309} C_VEL
LIN {X 0,Y 411.419,Z 504.838,A -85,B 0,C 180,E1 -10869.175,E2 -10869.175} C_VEL
LIN {X 0,Y 410.813,Z 519.039,A -85,B 0,C 180,E1 -10869.601,E2 -10869.601} C_VEL
LIN {X 0,Y 410.008,Z 533.257,A -85,B 0,C 180,E1 -10870.239,E2 -10870.239} C_VEL
LIN {X 0,Y 409.086,Z 547.047,A -85,B 0,C 180,E1 -10871.079,E2 -10871.079} C_VEL
LIN {X 0,Y 408.083,Z 559.737,A -85,B 0,C 180,E1 -10872.071,E2 -10872.071} C_VEL
LIN {X 0,Y 406.952,Z 571.293,A -85,B 0,C 180,E1 -10873.186,E2 -10873.186} C_VEL
LIN {X 0,Y 405.999,Z 581.904,A -85,B 0,C 180,E1 -10874.437,E2 -10874.437} C_VEL
LIN {X 0,Y 405.116,Z 592.444,A -85,B 0,C 180,E1 -10875.944,E2 -10875.944} C_VEL
LIN {X 0,Y 404.403,Z 601.131,A -85,B 0,C 180,E1 -10877.454,E2 -10877.454} C_VEL
LIN {X 0,Y 403.724,Z 609.438,A -85,B 0,C 180,E1 -10879.215,E2 -10879.215} C_VEL
LIN {X 0,Y 403.289,Z 616.111,A -85,B 0,C 180,E1 -10880.977,E2 -10880.977} C_VEL
LIN {X 0,Y 403.067,Z 622.03,A -85,B 0,C 180,E1 -10882.99,E2 -10882.99} C_VEL
LIN {X 0,Y 402.903,Z 626.352,A -85,B 0,C 180,E1 -10884.997,E2 -10884.997} C_VEL
LIN {X 0,Y 402.822,Z 629.215,A -85,B 0,C 180,E1 -10887,E2 -10887} C_VEL
LIN {X 0,Y 402.86,Z 630.705,A -85,B 0,C 180,E1 -10889,E2 -10889} C_VEL
LIN {X 0,Y 402.86,Z 630.851,A -85,B 0,C 180,E1 -10891,E2 -10891} C_VEL
LIN {X 0,Y 402.818,Z 629.666,A -85,B 0,C 180,E1 -10893,E2 -10893} C_VEL
LIN {X 0,Y 402.903,Z 627.132,A -85,B 0,C 180,E1 -10895.003,E2 -10895.003} C_VEL
LIN {X 0,Y 403.067,Z 623.159,A -85,B 0,C 180,E1 -10897.01,E2 -10897.01} C_VEL
LIN {X 0,Y 403.345,Z 617.63,A -85,B 0,C 180,E1 -10899.022,E2 -10899.022} C_VEL
LIN {X 0,Y 403.791,Z 611.405,A -85,B 0,C 180,E1 -10900.784,E2 -10900.784} C_VEL
LIN {X 0,Y 404.621,Z 603.664,A -85,B 0,C 180,E1 -10902.539,E2 -10902.539} C_VEL
LIN {X 0,Y 405.317,Z 595.603,A -85,B 0,C 180,E1 -10904.049,E2 -10904.049} C_VEL
LIN {X 0,Y 406.341,Z 585.907,A -85,B 0,C 180,E1 -10905.55,E2 -10905.55} C_VEL
LIN {X 0,Y 407.496,Z 575.166,A -85,B 0,C 180,E1 -10906.92,E2 -10906.92} C_VEL
LIN {X 0,Y 408.782,Z 563.292,A -85,B 0,C 180,E1 -10908.156,E2 -10908.156} C_VEL
LIN {X 0,Y 409.881,Z 551.787,A -85,B 0,C 180,E1 -10909.131,E2 -10909.131} C_VEL
LIN {X 0,Y 410.919,Z 538.966,A -85,B 0,C 180,E1 -10910.002,E2 -10910.002} C_VEL
LIN {X 0,Y 411.766,Z 526.096,A -85,B 0,C 180,E1 -10910.676,E2 -10910.676} C_VEL
LIN {X 0,Y 412.659,Z 511.492,A -85,B 0,C 180,E1 -10911.217,E2 -10911.217} C_VEL
LIN {X 0,Y 413.077,Z 496.943,A -85,B 0,C 180,E1 -10911.554,E2 -10911.554} C_VEL
LIN {X 0,Y 414.759,Z 399.127,A -85,B 0,C 180,E1 -10913.275,E2 -10913.275} C_VEL
LIN {X 0,Y 411.006,Z 378.832,A -85,B 0,C 180,E1 -10913.906,E2 -10913.906} C_VEL
LIN {X 0,Y 408.598,Z 367.199,A -85,B 0,C 180,E1 -10914.306,E2 -10914.306} C_VEL
LIN {X 0,Y 409.418,Z 357.116,A -85,B 0,C 180,E1 -10916.232,E2 -10916.232} C_VEL
LIN {X 0,Y 407.275,Z 346.336,A -85,B 0,C 180,E1 -10918.548,E2 -10918.548} C_VEL
LIN {X 0,Y 404.139,Z 333.771,A -85,B 0,C 180,E1 -10921.445,E2 -10921.445} C_VEL
LIN {X 0,Y 404.181,Z 333.763,A -85,B 0,C 180,E1 -10925.015,E2 -10925.015} C_VEL
LIN {X 0,Y 404.149,Z 333.764,A -85,B 0,C 180,E1 -10928.756,E2 -10928.756} C_VEL
LIN {X 0,Y 404.117,Z 333.763,A -85,B 0,C 180,E1 -10931.599,E2 -10931.599} C_VEL
LIN {X 0,Y 404.139,Z 333.764,A -85,B 0,C 180,E1 -10934.521,E2 -10934.521} C_VEL
LIN {X 0,Y 404.13,Z 333.764,A -85,B 0,C 180,E1 -10937.295,E2 -10937.295} C_VEL
LIN {X 0,Y 404.162,Z 333.764,A -85,B 0,C 180,E1 -10939.955,E2 -10939.955} C_VEL
LIN {X 0,Y 404.128,Z 333.767,A -85,B 0,C 180,E1 -10943.124,E2 -10943.124} C_VEL
LIN {X 0,Y 404.136,Z 333.77,A -85,B 0,C 180,E1 -10946.187,E2 -10946.187} C_VEL
LIN {X 0,Y 404.135,Z 333.75,A -85,B 0,C 180,E1 -10949.714,E2 -10949.714} C_VEL
LIN {X 0,Y 404.125,Z 333.767,A -85,B 0,C 180,E1 -10953.118,E2 -10953.118} C_VEL
LIN {X 0,Y 404.146,Z 333.766,A -85,B 0,C 180,E1 -10956.424,E2 -10956.424} C_VEL
LIN {X 0,Y 404.181,Z 333.76,A -85,B 0,C 180,E1 -10959.874,E2 -10959.874} C_VEL
LIN {X 0,Y 404.205,Z 333.757,A -85,B 0,C 180,E1 -10962.993,E2 -10962.993} C_VEL
LIN {X 0,Y 404.272,Z 333.75,A -85,B 0,C 180,E1 -10966.939,E2 -10966.939} C_VEL
LIN {X 0,Y 404.228,Z 333.758,A -85,B 0,C 180,E1 -10969.988,E2 -10969.988} C_VEL
LIN {X 0,Y 404.329,Z 333.738,A -85,B 0,C 180,E1 -10973.012,E2 -10973.012} C_VEL
LIN {X 0,Y 404.248,Z 333.753,A -85,B 0,C 180,E1 -10975.013,E2 -10975.013} C_VEL
LIN {X 0,Y 404.459,Z 333.722,A -85,B 0,C 180,E1 -10978.009,E2 -10978.009} C_VEL
LIN {X 0,Y 404.466,Z 333.72,A -85,B 0,C 180,E1 -10981.992,E2 -10981.992} C_VEL
LIN {X 0,Y 404.361,Z 333.735,A -85,B 0,C 180,E1 -10986.6,E2 -10986.6} C_VEL
LIN {X 0,Y 404.254,Z 333.753,A -85,B 0,C 180,E1 -10989.002,E2 -10989.002} C_VEL
LIN {X 0,Y 404.244,Z 333.745,A -85,B 0,C 180,E1 -10992.042,E2 -10992.042} C_VEL
LIN {X 0,Y 404.194,Z 333.762,A -85,B 0,C 180,E1 -10995.119,E2 -10995.119} C_VEL
LIN {X 0,Y 404.195,Z 333.759,A -85,B 0,C 180,E1 -10998.239,E2 -10998.239} C_VEL
LIN {X 0,Y 404.129,Z 333.769,A -85,B 0,C 180,E1 -11001.42,E2 -11001.42} C_VEL
LIN {X 0,Y 404.166,Z 333.762,A -85,B 0,C 180,E1 -11004.667,E2 -11004.667} C_VEL
LIN {X 0,Y 404.188,Z 333.757,A -85,B 0,C 180,E1 -11008.001,E2 -11008.001} C_VEL
LIN {X 0,Y 404.132,Z 333.764,A -85,B 0,C 180,E1 -11011.559,E2 -11011.559} C_VEL
LIN {X 0,Y 404.179,Z 333.763,A -85,B 0,C 180,E1 -11015.017,E2 -11015.017} C_VEL
LIN {X 0,Y 404.145,Z 333.769,A -85,B 0,C 180,E1 -11018.759,E2 -11018.759} C_VEL
LIN {X 0,Y 404.119,Z 333.769,A -85,B 0,C 180,E1 -11021.601,E2 -11021.601} C_VEL
LIN {X 0,Y 404.142,Z 333.768,A -85,B 0,C 180,E1 -11024.523,E2 -11024.523} C_VEL
LIN {X 0,Y 404.134,Z 333.769,A -85,B 0,C 180,E1 -11027.297,E2 -11027.297} C_VEL
LIN {X 0,Y 404.168,Z 333.768,A -85,B 0,C 180,E1 -11029.957,E2 -11029.957} C_VEL
LIN {X 0,Y 404.139,Z 333.768,A -85,B 0,C 180,E1 -11033.125,E2 -11033.125} C_VEL
LIN {X 0,Y 404.185,Z 333.891,A -85,B 0,C 180,E1 -11036.373,E2 -11036.373} C_VEL
LIN {X 0,Y 407.213,Z 347.037,A -85,B 0,C 180,E1 -11039.649,E2 -11039.649} C_VEL
LIN {X 0,Y 412.03,Z 359.065,A -85,B 0,C 180,E1 -11040.226,E2 -11040.226} C_VEL
LIN {X 0,Y 415.088,Z 372.633,A -85,B 0,C 180,E1 -11040.688,E2 -11040.688} C_VEL
LIN {X 0,Y 413.177,Z 483.339,A -85,B 0,C 180,E1 -11042.661,E2 -11042.661} C_VEL
LIN {X 0,Y 412.628,Z 497.511,A -85,B 0,C 180,E1 -11043.102,E2 -11043.102} C_VEL
LIN {X 0,Y 411.871,Z 511.291,A -85,B 0,C 180,E1 -11043.732,E2 -11043.732} C_VEL
LIN {X 0,Y 410.843,Z 524.643,A -85,B 0,C 180,E1 -11044.546,E2 -11044.546} C_VEL
LIN {X 0,Y 409.738,Z 537.624,A -85,B 0,C 180,E1 -11045.569,E2 -11045.569} C_VEL
LIN {X 0,Y 408.67,Z 547.94,A -85,B 0,C 180,E1 -11046.567,E2 -11046.567} C_VEL
LIN {X 0,Y 407.617,Z 557.797,A -85,B 0,C 180,E1 -11047.709,E2 -11047.709} C_VEL
LIN {X 0,Y 406.709,Z 567.483,A -85,B 0,C 180,E1 -11049.063,E2 -11049.063} C_VEL
LIN {X 0,Y 405.669,Z 576.227,A -85,B 0,C 180,E1 -11050.519,E2 -11050.519} C_VEL
LIN {X 0,Y 404.773,Z 584.988,A -85,B 0,C 180,E1 -11052.312,E2 -11052.312} C_VEL
LIN {X 0,Y 404.139,Z 591.115,A -85,B 0,C 180,E1 -11053.845,E2 -11053.845} C_VEL
LIN {X 0,Y 403.635,Z 596.165,A -85,B 0,C 180,E1 -11055.377,E2 -11055.377} C_VEL
LIN {X 0,Y 403.225,Z 601.385,A -85,B 0,C 180,E1 -11057.438,E2 -11057.438} C_VEL
LIN {X 0,Y 403.015,Z 604.236,A -85,B 0,C 180,E1 -11058.941,E2 -11058.941} C_VEL
LIN {X 0,Y 402.804,Z 606.801,A -85,B 0,C 180,E1 -11060.966,E2 -11060.966} C_VEL
LIN {X 0,Y 402.858,Z 607.988,A -85,B 0,C 180,E1 -11062.986,E2 -11062.986} C_VEL
LIN {X 0,Y 402.901,Z 608.082,A -85,B 0,C 180,E1 -11064,E2 -11064} C_VEL
LIN {X 0,Y 402.187,Z 607.948,A -85,B 0,C 180,E1 -11064.834,E2 -11064.834} C_VEL
LIN {X 0,Y 399.33,Z 607.241,A -85,B 0,C 180,E1 -11066.187,E2 -11066.187} C_VEL
LIN {X 0,Y 396.949,Z 606.281,A -85,B 0,C 180,E1 -11067.274,E2 -11067.274} C_VEL
LIN {X 0,Y 395.936,Z 605.267,A -85,B 0,C 180,E1 -11068.107,E2 -11068.107} C_VEL
LIN {X 0,Y 395.856,Z 604.829,A -85,B 0,C 180,E1 -11068.387,E2 -11068.387} C_VEL
LIN {X 0,Y 396.041,Z 600.968,A -85,B 0,C 180,E1 -11070.508,E2 -11070.508} C_VEL
LIN {X 0,Y 396.386,Z 595.643,A -85,B 0,C 180,E1 -11072.54,E2 -11072.54} C_VEL
LIN {X 0,Y 396.7,Z 590.566,A -85,B 0,C 180,E1 -11074.064,E2 -11074.064} C_VEL
LIN {X 0,Y 397.483,Z 583.284,A -85,B 0,C 180,E1 -11075.835,E2 -11075.835} C_VEL
LIN {X 0,Y 398.428,Z 574.245,A -85,B 0,C 180,E1 -11077.602,E2 -11077.602} C_VEL
LIN {X 0,Y 399.239,Z 564.82,A -85,B 0,C 180,E1 -11079.116,E2 -11079.116} C_VEL
LIN {X 0,Y 400.273,Z 553.747,A -85,B 0,C 180,E1 -11080.572,E2 -11080.572} C_VEL
LIN {X 0,Y 401.479,Z 541.561,A -85,B 0,C 180,E1 -11081.869,E2 -11081.869} C_VEL
LIN {X 0,Y 402.389,Z 530.043,A -85,B 0,C 180,E1 -11082.867,E2 -11082.867} C_VEL
LIN {X 0,Y 403.373,Z 516.526,A -85,B 0,C 180,E1 -11083.796,E2 -11083.796} C_VEL
LIN {X 0,Y 404.169,Z 503.504,A -85,B 0,C 180,E1 -11084.475,E2 -11084.475} C_VEL
LIN {X 0,Y 404.821,Z 489.442,A -85,B 0,C 180,E1 -11084.997,E2 -11084.997} C_VEL
LIN {X 0,Y 405.098,Z 474.758,A -85,B 0,C 180,E1 -11085.341,E2 -11085.341} C_VEL
LIN {X 0,Y 406.572,Z 372.569,A -85,B 0,C 180,E1 -11087.156,E2 -11087.156} C_VEL
LIN {X 0,Y 402.767,Z 355.365,A -85,B 0,C 180,E1 -11087.691,E2 -11087.691} C_VEL
LIN {X 0,Y 399.753,Z 347.011,A -85,B 0,C 180,E1 -11088.04,E2 -11088.04} C_VEL
LIN {X 0,Y 397.124,Z 334.647,A -85,B 0,C 180,E1 -11090.999,E2 -11090.999} C_VEL
LIN {X 0,Y 397.135,Z 334.644,A -85,B 0,C 180,E1 -11094.017,E2 -11094.017} C_VEL
LIN {X 0,Y 397.196,Z 334.635,A -85,B 0,C 180,E1 -11097.389,E2 -11097.389} C_VEL
LIN {X 0,Y 397.079,Z 334.646,A -85,B 0,C 180,E1 -11100.881,E2 -11100.881} C_VEL
LIN {X 0,Y 397.126,Z 334.638,A -85,B 0,C 180,E1 -11104.492,E2 -11104.492} C_VEL
LIN {X 0,Y 397.105,Z 334.642,A -85,B 0,C 180,E1 -11108.273,E2 -11108.273} C_VEL
LIN {X 0,Y 397.087,Z 334.632,A -85,B 0,C 180,E1 -11110.908,E2 -11110.908} C_VEL
LIN {X 0,Y 397.098,Z 334.646,A -85,B 0,C 180,E1 -11113.647,E2 -11113.647} C_VEL
LIN {X 0,Y 397.098,Z 334.643,A -85,B 0,C 180,E1 -11116.52,E2 -11116.52} C_VEL
LIN {X 0,Y 397.108,Z 334.642,A -85,B 0,C 180,E1 -11120.421,E2 -11120.421} C_VEL
LIN {X 0,Y 397.102,Z 334.643,A -85,B 0,C 180,E1 -11124.264,E2 -11124.264} C_VEL
LIN {X 0,Y 397.108,Z 334.64,A -85,B 0,C 180,E1 -11126.726,E2 -11126.726} C_VEL
LIN {X 0,Y 397.117,Z 334.64,A -85,B 0,C 180,E1 -11130.295,E2 -11130.295} C_VEL
LIN {X 0,Y 397.186,Z 334.623,A -85,B 0,C 180,E1 -11132.609,E2 -11132.609} C_VEL
LIN {X 0,Y 397.114,Z 334.641,A -85,B 0,C 180,E1 -11135.98,E2 -11135.98} C_VEL
LIN {X 0,Y 397.13,Z 334.626,A -85,B 0,C 180,E1 -11139.704,E2 -11139.704} C_VEL
LIN {X 0,Y 397.173,Z 334.637,A -85,B 0,C 180,E1 -11142.844,E2 -11142.844} C_VEL
LIN {X 0,Y 397.219,Z 334.618,A -85,B 0,C 180,E1 -11146.702,E2 -11146.702} C_VEL
LIN {X 0,Y 397.203,Z 334.627,A -85,B 0,C 180,E1 -11149.808,E2 -11149.808} C_VEL
LIN {X 0,Y 397.319,Z 334.614,A -85,B 0,C 180,E1 -11152.887,E2 -11152.887} C_VEL
LIN {X 0,Y 397.229,Z 334.613,A -85,B 0,C 180,E1 -11154.924,E2 -11154.924} C_VEL
LIN {X 0,Y 397.431,Z 334.598,A -85,B 0,C 180,E1 -11157.973,E2 -11157.973} C_VEL
LIN {X 0,Y 397.423,Z 334.601,A -85,B 0,C 180,E1 -11162.027,E2 -11162.027} C_VEL
LIN {X 0,Y 397.308,Z 334.619,A -85,B 0,C 180,E1 -11166.092,E2 -11166.092} C_VEL
LIN {X 0,Y 397.218,Z 334.619,A -85,B 0,C 180,E1 -11169.162,E2 -11169.162} C_VEL
LIN {X 0,Y 397.206,Z 334.634,A -85,B 0,C 180,E1 -11172.258,E2 -11172.258} C_VEL
LIN {X 0,Y 397.166,Z 334.627,A -85,B 0,C 180,E1 -11175.392,E2 -11175.392} C_VEL
LIN {X 0,Y 397.146,Z 334.638,A -85,B 0,C 180,E1 -11178.574,E2 -11178.574} C_VEL
LIN {X 0,Y 397.085,Z 334.638,A -85,B 0,C 180,E1 -11181.819,E2 -11181.819} C_VEL
LIN {X 0,Y 397.113,Z 334.637,A -85,B 0,C 180,E1 -11185.134,E2 -11185.134} C_VEL
LIN {X 0,Y 397.069,Z 334.647,A -85,B 0,C 180,E1 -11188.548,E2 -11188.548} C_VEL
LIN {X 0,Y 397.073,Z 334.649,A -85,B 0,C 180,E1 -11191.837,E2 -11191.837} C_VEL
LIN {X 0,Y 397.117,Z 334.641,A -85,B 0,C 180,E1 -11194.494,E2 -11194.494} C_VEL
LIN {X 0,Y 397.096,Z 334.646,A -85,B 0,C 180,E1 -11198.276,E2 -11198.276} C_VEL
LIN {X 0,Y 397.081,Z 334.639,A -85,B 0,C 180,E1 -11200.909,E2 -11200.909} C_VEL
LIN {X 0,Y 397.094,Z 334.648,A -85,B 0,C 180,E1 -11203.649,E2 -11203.649} C_VEL
LIN {X 0,Y 397.096,Z 334.643,A -85,B 0,C 180,E1 -11206.522,E2 -11206.522} C_VEL
LIN {X 0,Y 397.107,Z 334.646,A -85,B 0,C 180,E1 -11210.423,E2 -11210.423} C_VEL
LIN {X 0,Y 397.104,Z 334.648,A -85,B 0,C 180,E1 -11214.266,E2 -11214.266} C_VEL
LIN {X 0,Y 397.111,Z 334.646,A -85,B 0,C 180,E1 -11216.728,E2 -11216.728} C_VEL
LIN {X 0,Y 397.139,Z 334.746,A -85,B 0,C 180,E1 -11219.403,E2 -11219.403} C_VEL
LIN {X 0,Y 400.147,Z 347.977,A -85,B 0,C 180,E1 -11222.263,E2 -11222.263} C_VEL
LIN {X 0,Y 401.682,Z 356.682,A -85,B 0,C 180,E1 -11224.062,E2 -11224.062} C_VEL
LIN {X 0,Y 400.833,Z 367.222,A -85,B 0,C 180,E1 -11226.054,E2 -11226.054} C_VEL
LIN {X 0,Y 406.342,Z 400.215,A -85,B 0,C 180,E1 -11226.983,E2 -11226.983} C_VEL
LIN {X 0,Y 404.689,Z 504.468,A -85,B 0,C 180,E1 -11228.845,E2 -11228.845} C_VEL
LIN {X 0,Y 404.105,Z 518.757,A -85,B 0,C 180,E1 -11229.28,E2 -11229.28} C_VEL
LIN {X 0,Y 403.279,Z 532.425,A -85,B 0,C 180,E1 -11229.895,E2 -11229.895} C_VEL
LIN {X 0,Y 402.367,Z 546.101,A -85,B 0,C 180,E1 -11230.732,E2 -11230.732} C_VEL
LIN {X 0,Y 401.251,Z 559.139,A -85,B 0,C 180,E1 -11231.755,E2 -11231.755} C_VEL
LIN {X 0,Y 400.133,Z 570.771,A -85,B 0,C 180,E1 -11232.891,E2 -11232.891} C_VEL
LIN {X 0,Y 399.108,Z 581.436,A -85,B 0,C 180,E1 -11234.161,E2 -11234.161} C_VEL
LIN {X 0,Y 398.161,Z 592.02,A -85,B 0,C 180,E1 -11235.694,E2 -11235.694} C_VEL
LIN {X 0,Y 397.438,Z 600.747,A -85,B 0,C 180,E1 -11237.23,E2 -11237.23} C_VEL
LIN {X 0,Y 396.709,Z 609.099,A -85,B 0,C 180,E1 -11239.022,E2 -11239.022} C_VEL
LIN {X 0,Y 396.243,Z 615.802,A -85,B 0,C 180,E1 -11240.815,E2 -11240.815} C_VEL
LIN {X 0,Y 395.986,Z 621.747,A -85,B 0,C 180,E1 -11242.864,E2 -11242.864} C_VEL
LIN {X 0,Y 395.822,Z 626.092,A -85,B 0,C 180,E1 -11244.907,E2 -11244.907} C_VEL
LIN {X 0,Y 395.725,Z 628.977,A -85,B 0,C 180,E1 -11246.946,E2 -11246.946} C_VEL
LIN {X 0,Y 395.789,Z 630.488,A -85,B 0,C 180,E1 -11248.983,E2 -11248.983} C_VEL
LIN {X 0,Y 395.789,Z 630.655,A -85,B 0,C 180,E1 -11251.017,E2 -11251.017} C_VEL
LIN {X 0,Y 395.721,Z 629.489,A -85,B 0,C 180,E1 -11253.054,E2 -11253.054} C_VEL
LIN {X 0,Y 395.802,Z 626.978,A -85,B 0,C 180,E1 -11255.093,E2 -11255.093} C_VEL
LIN {X 0,Y 395.99,Z 623.037,A -85,B 0,C 180,E1 -11257.136,E2 -11257.136} C_VEL
LIN {X 0,Y 396.299,Z 617.534,A -85,B 0,C 180,E1 -11259.184,E2 -11259.184} C_VEL
LIN {X 0,Y 396.791,Z 611.337,A -85,B 0,C 180,E1 -11260.976,E2 -11260.976} C_VEL
LIN {X 0,Y 397.629,Z 603.626,A -85,B 0,C 180,E1 -11262.764,E2 -11262.764} C_VEL
LIN {X 0,Y 398.402,Z 595.602,A -85,B 0,C 180,E1 -11264.298,E2 -11264.298} C_VEL
LIN {X 0,Y 399.484,Z 585.948,A -85,B 0,C 180,E1 -11265.824,E2 -11265.824} C_VEL
LIN {X 0,Y 400.685,Z 575.258,A -85,B 0,C 180,E1 -11267.216,E2 -11267.216} C_VEL
LIN {X 0,Y 402.04,Z 563.447,A -85,B 0,C 180,E1 -11268.471,E2 -11268.471} C_VEL
LIN {X 0,Y 403.288,Z 551.136,A -85,B 0,C 180,E1 -11269.53,E2 -11269.53} C_VEL
LIN {X 0,Y 404.366,Z 538.327,A -85,B 0,C 180,E1 -11270.407,E2 -11270.407} C_VEL
LIN {X 0,Y 405.262,Z 525.325,A -85,B 0,C 180,E1 -11271.09,E2 -11271.09} C_VEL
LIN {X 0,Y 406.143,Z 511.418,A -85,B 0,C 180,E1 -11271.607,E2 -11271.607} C_VEL
LIN {X 0,Y 406.584,Z 496.968,A -85,B 0,C 180,E1 -11271.949,E2 -11271.949} C_VEL
LIN {X 0,Y 408.335,Z 400.788,A -85,B 0,C 180,E1 -11273.666,E2 -11273.666} C_VEL
LIN {X 0,Y 405.744,Z 385.384,A -85,B 0,C 180,E1 -11274.138,E2 -11274.138} C_VEL
LIN {X 0,Y 401.869,Z 367.021,A -85,B 0,C 180,E1 -11274.776,E2 -11274.776} C_VEL
LIN {X 0,Y 402.548,Z 358.568,A -85,B 0,C 180,E1 -11276.424,E2 -11276.424} C_VEL
LIN {X 0,Y 400.505,Z 348.321,A -85,B 0,C 180,E1 -11278.671,E2 -11278.671} C_VEL
LIN {X 0,Y 397.096,Z 334.649,A -85,B 0,C 180,E1 -11281.862,E2 -11281.862} C_VEL
LIN {X 0,Y 397.122,Z 334.645,A -85,B 0,C 180,E1 -11284.493,E2 -11284.493} C_VEL
LIN {X 0,Y 397.098,Z 334.64,A -85,B 0,C 180,E1 -11288.274,E2 -11288.274} C_VEL
LIN {X 0,Y 397.083,Z 334.637,A -85,B 0,C 180,E1 -11290.908,E2 -11290.908} C_VEL
LIN {X 0,Y 397.095,Z 334.639,A -85,B 0,C 180,E1 -11293.648,E2 -11293.648} C_VEL
LIN {X 0,Y 397.096,Z 334.644,A -85,B 0,C 180,E1 -11296.52,E2 -11296.52} C_VEL
LIN {X 0,Y 397.106,Z 334.646,A -85,B 0,C 180,E1 -11300.422,E2 -11300.422} C_VEL
LIN {X 0,Y 397.1,Z 334.645,A -85,B 0,C 180,E1 -11304.265,E2 -11304.265} C_VEL
LIN {X 0,Y 397.106,Z 334.643,A -85,B 0,C 180,E1 -11306.726,E2 -11306.726} C_VEL
LIN {X 0,Y 397.109,Z 334.624,A -85,B 0,C 180,E1 -11310.295,E2 -11310.295} C_VEL
LIN {X 0,Y 397.085,Z 334.649,A -85,B 0,C 180,E1 -11313.738,E2 -11313.738} C_VEL
LIN {X 0,Y 397.092,Z 334.644,A -85,B 0,C 180,E1 -11317.085,E2 -11317.085} C_VEL
LIN {X 0,Y 397.135,Z 334.639,A -85,B 0,C 180,E1 -11320.352,E2 -11320.352} C_VEL
LIN {X 0,Y 397.155,Z 334.634,A -85,B 0,C 180,E1 -11323.553,E2 -11323.553} C_VEL
LIN {X 0,Y 397.218,Z 334.628,A -85,B 0,C 180,E1 -11326.703,E2 -11326.703} C_VEL
LIN {X 0,Y 397.19,Z 334.636,A -85,B 0,C 180,E1 -11329.809,E2 -11329.809} C_VEL
LIN {X 0,Y 397.282,Z 334.616,A -85,B 0,C 180,E1 -11332.887,E2 -11332.887} C_VEL
LIN {X 0,Y 397.22,Z 334.628,A -85,B 0,C 180,E1 -11334.925,E2 -11334.925} C_VEL
LIN {X 0,Y 397.428,Z 334.598,A -85,B 0,C 180,E1 -11337.974,E2 -11337.974} C_VEL
LIN {X 0,Y 397.434,Z 334.596,A -85,B 0,C 180,E1 -11342.027,E2 -11342.027} C_VEL
LIN {X 0,Y 397.312,Z 334.613,A -85,B 0,C 180,E1 -11346.597,E2 -11346.597} C_VEL
LIN {X 0,Y 397.224,Z 334.63,A -85,B 0,C 180,E1 -11349.163,E2 -11349.163} C_VEL
LIN {X 0,Y 397.207,Z 334.622,A -85,B 0,C 180,E1 -11352.259,E2 -11352.259} C_VEL
LIN {X 0,Y 397.168,Z 334.633,A -85,B 0,C 180,E1 -11355.393,E2 -11355.393} C_VEL
LIN {X 0,Y 397.148,Z 334.639,A -85,B 0,C 180,E1 -11358.575,E2 -11358.575} C_VEL
LIN {X 0,Y 397.087,Z 334.644,A -85,B 0,C 180,E1 -11361.82,E2 -11361.82} C_VEL
LIN {X 0,Y 397.145,Z 334.638,A -85,B 0,C 180,E1 -11365.513,E2 -11365.513} C_VEL
LIN {X 0,Y 397.115,Z 334.64,A -85,B 0,C 180,E1 -11368.545,E2 -11368.545} C_VEL
LIN {X 0,Y 397.072,Z 334.644,A -85,B 0,C 180,E1 -11372.073,E2 -11372.073} C_VEL
LIN {X 0,Y 397.114,Z 334.641,A -85,B 0,C 180,E1 -11375.504,E2 -11375.504} C_VEL
LIN {X 0,Y 397.122,Z 334.642,A -85,B 0,C 180,E1 -11378.862,E2 -11378.862} C_VEL
LIN {X 0,Y 397.065,Z 334.649,A -85,B 0,C 180,E1 -11382.268,E2 -11382.268} C_VEL
LIN {X 0,Y 397.084,Z 334.648,A -85,B 0,C 180,E1 -11385.07,E2 -11385.07} C_VEL
LIN {X 0,Y 397.065,Z 334.652,A -85,B 0,C 180,E1 -11388.022,E2 -11388.022} C_VEL
LIN {X 0,Y 397.133,Z 334.642,A -85,B 0,C 180,E1 -11391.139,E2 -11391.139} C_VEL
LIN {X 0,Y 397.12,Z 334.641,A -85,B 0,C 180,E1 -11394.498,E2 -11394.498} C_VEL
LIN {X 0,Y 397.131,Z 334.733,A -85,B 0,C 180,E1 -11395.94,E2 -11395.94} C_VEL
LIN {X 0,Y 400.121,Z 347.495,A -85,B 0,C 180,E1 -11399.159,E2 -11399.159} C_VEL
LIN {X 0,Y 405.953,Z 361.57,A -85,B 0,C 180,E1 -11399.854,E2 -11399.854} C_VEL
LIN {X 0,Y 408.686,Z 373.805,A -85,B 0,C 180,E1 -11400.28,E2 -11400.28} C_VEL
LIN {X 0,Y 406.695,Z 483.244,A -85,B 0,C 180,E1 -11402.258,E2 -11402.258} C_VEL
LIN {X 0,Y 406.121,Z 497.541,A -85,B 0,C 180,E1 -11402.705,E2 -11402.705} C_VEL
LIN {X 0,Y 405.315,Z 511.361,A -85,B 0,C 180,E1 -11403.343,E2 -11403.343} C_VEL
LIN {X 0,Y 404.324,Z 523.843,A -85,B 0,C 180,E1 -11404.106,E2 -11404.106} C_VEL
LIN {X 0,Y 403.179,Z 536.888,A -85,B 0,C 180,E1 -11405.133,E2 -11405.133} C_VEL
LIN {X 0,Y 402.023,Z 547.473,A -85,B 0,C 180,E1 -11406.156,E2 -11406.156} C_VEL
LIN {X 0,Y 400.686,Z 559.418,A -85,B 0,C 180,E1 -11407.574,E2 -11407.574} C_VEL
LIN {X 0,Y 399.663,Z 569.458,A -85,B 0,C 180,E1 -11409.043,E2 -11409.043} C_VEL
LIN {X 0,Y 398.527,Z 578.776,A -85,B 0,C 180,E1 -11410.692,E2 -11410.692} C_VEL
LIN {X 0,Y 397.608,Z 587.095,A -85,B 0,C 180,E1 -11412.514,E2 -11412.514} C_VEL
LIN {X 0,Y 396.986,Z 592.877,A -85,B 0,C 180,E1 -11414.074,E2 -11414.074} C_VEL
LIN {X 0,Y 396.499,Z 597.593,A -85,B 0,C 180,E1 -11415.632,E2 -11415.632} C_VEL
LIN {X 0,Y 396.116,Z 602.457,A -85,B 0,C 180,E1 -11417.708,E2 -11417.708} C_VEL
LIN {X 0,Y 395.775,Z 605.803,A -85,B 0,C 180,E1 -11419.772,E2 -11419.772} C_VEL
LIN {X 0,Y 395.751,Z 607.727,A -85,B 0,C 180,E1 -11421.833,E2 -11421.833} C_VEL
LIN {X 0,Y 395.815,Z 608.276,A -85,B 0,C 180,E1 -11423.988,E2 -11423.988} C_VEL
LIN {X 0,Y 395.76,Z 607.549,A -85,B 0,C 180,E1 -11425.927,E2 -11425.927} C_VEL
LIN {X 0,Y 395.867,Z 605.47,A -85,B 0,C 180,E1 -11427.965,E2 -11427.965} C_VEL
LIN {X 0,Y 395.856,Z 604.829,A -85,B 0,C 180,E1 -11428.387,E2 -11428.387} C_VEL
LIN {X 0,Y 395.236,Z 603.558,A -85,B 0,C 180,E1 -11429.217,E2 -11429.217} C_VEL
LIN {X 0,Y 392.562,Z 601.07,A -85,B 0,C 180,E1 -11430.559,E2 -11430.559} C_VEL
LIN {X 0,Y 390.319,Z 598.693,A -85,B 0,C 180,E1 -11431.622,E2 -11431.622} C_VEL
LIN {X 0,Y 389.382,Z 596.547,A -85,B 0,C 180,E1 -11432.424,E2 -11432.424} C_VEL
LIN {X 0,Y 389.319,Z 595.751,A -85,B 0,C 180,E1 -11432.69,E2 -11432.69} C_VEL
LIN {X 0,Y 389.84,Z 589.1,A -85,B 0,C 180,E1 -11434.653,E2 -11434.653} C_VEL
LIN {X 0,Y 390.739,Z 581.404,A -85,B 0,C 180,E1 -11436.454,E2 -11436.454} C_VEL
LIN {X 0,Y 391.551,Z 573.391,A -85,B 0,C 180,E1 -11437.996,E2 -11437.996} C_VEL
LIN {X 0,Y 392.433,Z 564.091,A -85,B 0,C 180,E1 -11439.485,E2 -11439.485} C_VEL
LIN {X 0,Y 393.468,Z 553.374,A -85,B 0,C 180,E1 -11440.901,E2 -11440.901} C_VEL
LIN {X 0,Y 394.594,Z 542.473,A -85,B 0,C 180,E1 -11442.08,E2 -11442.08} C_VEL
LIN {X 0,Y 395.528,Z 531.114,A -85,B 0,C 180,E1 -11443.094,E2 -11443.094} C_VEL
LIN {X 0,Y 396.456,Z 518.803,A -85,B 0,C 180,E1 -11443.977,E2 -11443.977} C_VEL
LIN {X 0,Y 397.366,Z 505.132,A -85,B 0,C 180,E1 -11444.728,E2 -11444.728} C_VEL
LIN {X 0,Y 398.081,Z 490.85,A -85,B 0,C 180,E1 -11445.29,E2 -11445.29} C_VEL
LIN {X 0,Y 398.408,Z 477.063,A -85,B 0,C 180,E1 -11445.638,E2 -11445.638} C_VEL
LIN {X 0,Y 399.982,Z 373.943,A -85,B 0,C 180,E1 -11447.498,E2 -11447.498} C_VEL
LIN {X 0,Y 396.448,Z 357.642,A -85,B 0,C 180,E1 -11448.012,E2 -11448.012} C_VEL
LIN {X 0,Y 392.625,Z 347.255,A -85,B 0,C 180,E1 -11448.45,E2 -11448.45} C_VEL
LIN {X 0,Y 390.056,Z 335.526,A -85,B 0,C 180,E1 -11451.329,E2 -11451.329} C_VEL
LIN {X 0,Y 390.082,Z 335.52,A -85,B 0,C 180,E1 -11454.48,E2 -11454.48} C_VEL
LIN {X 0,Y 390.119,Z 335.515,A -85,B 0,C 180,E1 -11457.929,E2 -11457.929} C_VEL
LIN {X 0,Y 390.025,Z 335.528,A -85,B 0,C 180,E1 -11461.503,E2 -11461.503} C_VEL
LIN {X 0,Y 390.086,Z 335.514,A -85,B 0,C 180,E1 -11465.206,E2 -11465.206} C_VEL
LIN {X 0,Y 390.09,Z 335.517,A -85,B 0,C 180,E1 -11469.091,E2 -11469.091} C_VEL
LIN {X 0,Y 390.04,Z 335.521,A -85,B 0,C 180,E1 -11472.373,E2 -11472.373} C_VEL
LIN {X 0,Y 390.041,Z 335.523,A -85,B 0,C 180,E1 -11475.353,E2 -11475.353} C_VEL
LIN {X 0,Y 390.026,Z 335.519,A -85,B 0,C 180,E1 -11478.185,E2 -11478.185} C_VEL
LIN {X 0,Y 390.083,Z 335.52,A -85,B 0,C 180,E1 -11480.906,E2 -11480.906} C_VEL
LIN {X 0,Y 390.079,Z 335.52,A -85,B 0,C 180,E1 -11484.792,E2 -11484.792} C_VEL
LIN {X 0,Y 390.016,Z 335.525,A -85,B 0,C 180,E1 -11488.494,E2 -11488.494} C_VEL
LIN {X 0,Y 390.111,Z 335.503,A -85,B 0,C 180,E1 -11492.069,E2 -11492.069} C_VEL
LIN {X 0,Y 390.053,Z 335.522,A -85,B 0,C 180,E1 -11495.517,E2 -11495.517} C_VEL
LIN {X 0,Y 390.046,Z 335.513,A -85,B 0,C 180,E1 -11498.877,E2 -11498.877} C_VEL
LIN {X 0,Y 390.102,Z 335.512,A -85,B 0,C 180,E1 -11502.165,E2 -11502.165} C_VEL
LIN {X 0,Y 390.133,Z 335.505,A -85,B 0,C 180,E1 -11505.392,E2 -11505.392} C_VEL
LIN {X 0,Y 390.133,Z 335.501,A -85,B 0,C 180,E1 -11508.57,E2 -11508.57} C_VEL
LIN {X 0,Y 390.259,Z 335.495,A -85,B 0,C 180,E1 -11512.071,E2 -11512.071} C_VEL
LIN {X 0,Y 390.2,Z 335.489,A -85,B 0,C 180,E1 -11514.833,E2 -11514.833} C_VEL
LIN {X 0,Y 390.398,Z 335.474,A -85,B 0,C 180,E1 -11517.936,E2 -11517.936} C_VEL
LIN {X 0,Y 390.39,Z 335.477,A -85,B 0,C 180,E1 -11522.063,E2 -11522.063} C_VEL
LIN {X 0,Y 390.263,Z 335.498,A -85,B 0,C 180,E1 -11526.203,E2 -11526.203} C_VEL
LIN {X 0,Y 390.177,Z 335.495,A -85,B 0,C 180,E1 -11529.329,E2 -11529.329} C_VEL
LIN {X 0,Y 390.158,Z 335.512,A -85,B 0,C 180,E1 -11532.483,E2 -11532.483} C_VEL
LIN {X 0,Y 390.127,Z 335.505,A -85,B 0,C 180,E1 -11535.677,E2 -11535.677} C_VEL
LIN {X 0,Y 390.091,Z 335.515,A -85,B 0,C 180,E1 -11538.923,E2 -11538.923} C_VEL
LIN {X 0,Y 390.027,Z 335.522,A -85,B 0,C 180,E1 -11542.235,E2 -11542.235} C_VEL
LIN {X 0,Y 390.057,Z 335.518,A -85,B 0,C 180,E1 -11545.728,E2 -11545.728} C_VEL
LIN {X 0,Y 390.023,Z 335.523,A -85,B 0,C 180,E1 -11549.112,E2 -11549.112} C_VEL
LIN {X 0,Y 390.034,Z 335.523,A -85,B 0,C 180,E1 -11552.722,E2 -11552.722} C_VEL
LIN {X 0,Y 390.048,Z 335.527,A -85,B 0,C 180,E1 -11555.826,E2 -11555.826} C_VEL
LIN {X 0,Y 390.063,Z 335.521,A -85,B 0,C 180,E1 -11559.219,E2 -11559.219} C_VEL
LIN {X 0,Y 390.036,Z 335.521,A -85,B 0,C 180,E1 -11562.375,E2 -11562.375} C_VEL
LIN {X 0,Y 390.038,Z 335.524,A -85,B 0,C 180,E1 -11565.355,E2 -11565.355} C_VEL
LIN {X 0,Y 390.025,Z 335.526,A -85,B 0,C 180,E1 -11568.187,E2 -11568.187} C_VEL
LIN {X 0,Y 390.082,Z 335.522,A -85,B 0,C 180,E1 -11570.908,E2 -11570.908} C_VEL
LIN {X 0,Y 390.081,Z 335.524,A -85,B 0,C 180,E1 -11574.794,E2 -11574.794} C_VEL
LIN {X 0,Y 390.035,Z 335.527,A -85,B 0,C 180,E1 -11578.498,E2 -11578.498} C_VEL
LIN {X 0,Y 390.095,Z 335.647,A -85,B 0,C 180,E1 -11579.069,E2 -11579.069} C_VEL
LIN {X 0,Y 393.196,Z 349.154,A -85,B 0,C 180,E1 -11582.053,E2 -11582.053} C_VEL
LIN {X 0,Y 394.751,Z 357.685,A -85,B 0,C 180,E1 -11583.856,E2 -11583.856} C_VEL
LIN {X 0,Y 393.991,Z 367.287,A -85,B 0,C 180,E1 -11585.667,E2 -11585.667} C_VEL
LIN {X 0,Y 399.712,Z 401.118,A -85,B 0,C 180,E1 -11586.639,E2 -11586.639} C_VEL
LIN {X 0,Y 397.969,Z 505.37,A -85,B 0,C 180,E1 -11588.539,E2 -11588.539} C_VEL
LIN {X 0,Y 397.284,Z 519.983,A -85,B 0,C 180,E1 -11589.009,E2 -11589.009} C_VEL
LIN {X 0,Y 396.39,Z 534.549,A -85,B 0,C 180,E1 -11589.707,E2 -11589.707} C_VEL
LIN {X 0,Y 395.493,Z 546.757,A -85,B 0,C 180,E1 -11590.487,E2 -11590.487} C_VEL
LIN {X 0,Y 394.326,Z 559.972,A -85,B 0,C 180,E1 -11591.558,E2 -11591.558} C_VEL
LIN {X 0,Y 393.173,Z 571.423,A -85,B 0,C 180,E1 -11592.713,E2 -11592.713} C_VEL
LIN {X 0,Y 392.019,Z 582.923,A -85,B 0,C 180,E1 -11594.134,E2 -11594.134} C_VEL
LIN {X 0,Y 391.061,Z 593.235,A -85,B 0,C 180,E1 -11595.705,E2 -11595.705} C_VEL
LIN {X 0,Y 390.317,Z 601.673,A -85,B 0,C 180,E1 -11597.258,E2 -11597.258} C_VEL
LIN {X 0,Y 389.71,Z 608.754,A -85,B 0,C 180,E1 -11598.822,E2 -11598.822} C_VEL
LIN {X 0,Y 389.169,Z 615.489,A -85,B 0,C 180,E1 -11600.646,E2 -11600.646} C_VEL
LIN {X 0,Y 388.91,Z 621.461,A -85,B 0,C 180,E1 -11602.733,E2 -11602.733} C_VEL
LIN {X 0,Y 388.726,Z 625.83,A -85,B 0,C 180,E1 -11604.814,E2 -11604.814} C_VEL
LIN {X 0,Y 388.632,Z 628.738,A -85,B 0,C 180,E1 -11606.89,E2 -11606.89} C_VEL
LIN {X 0,Y 388.701,Z 630.271,A -85,B 0,C 180,E1 -11608.964,E2 -11608.964} C_VEL
LIN {X 0,Y 388.701,Z 630.459,A -85,B 0,C 180,E1 -11611.036,E2 -11611.036} C_VEL
LIN {X 0,Y 388.628,Z 629.314,A -85,B 0,C 180,E1 -11613.11,E2 -11613.11} C_VEL
LIN {X 0,Y 388.706,Z 626.824,A -85,B 0,C 180,E1 -11615.187,E2 -11615.187} C_VEL
LIN {X 0,Y 388.916,Z 622.916,A -85,B 0,C 180,E1 -11617.267,E2 -11617.267} C_VEL
LIN {X 0,Y 389.266,Z 617.441,A -85,B 0,C 180,E1 -11619.351,E2 -11619.351} C_VEL
LIN {X 0,Y 389.772,Z 611.272,A -85,B 0,C 180,E1 -11621.176,E2 -11621.176} C_VEL
LIN {X 0,Y 390.641,Z 603.594,A -85,B 0,C 180,E1 -11622.996,E2 -11622.996} C_VEL
LIN {X 0,Y 391.472,Z 595.606,A -85,B 0,C 180,E1 -11624.556,E2 -11624.556} C_VEL
LIN {X 0,Y 392.62,Z 585.995,A -85,B 0,C 180,E1 -11626.108,E2 -11626.108} C_VEL
LIN {X 0,Y 393.892,Z 575.358,A -85,B 0,C 180,E1 -11627.523,E2 -11627.523} C_VEL
LIN {X 0,Y 395.306,Z 563.611,A -85,B 0,C 180,E1 -11628.798,E2 -11628.798} C_VEL
LIN {X 0,Y 396.664,Z 550.691,A -85,B 0,C 180,E1 -11629.93,E2 -11629.93} C_VEL
LIN {X 0,Y 397.802,Z 537.703,A -85,B 0,C 180,E1 -11630.827,E2 -11630.827} C_VEL
LIN {X 0,Y 398.805,Z 524.558,A -85,B 0,C 180,E1 -11631.516,E2 -11631.516} C_VEL
LIN {X 0,Y 399.676,Z 510.288,A -85,B 0,C 180,E1 -11632.043,E2 -11632.043} C_VEL
LIN {X 0,Y 400.142,Z 495.266,A -85,B 0,C 180,E1 -11632.39,E2 -11632.39} C_VEL
LIN {X 0,Y 401.879,Z 400.664,A -85,B 0,C 180,E1 -11634.109,E2 -11634.109} C_VEL
LIN {X 0,Y 397.502,Z 377.65,A -85,B 0,C 180,E1 -11634.873,E2 -11634.873} C_VEL
LIN {X 0,Y 395.175,Z 366.824,A -85,B 0,C 180,E1 -11635.266,E2 -11635.266} C_VEL
LIN {X 0,Y 395.726,Z 360.288,A -85,B 0,C 180,E1 -11636.565,E2 -11636.565} C_VEL
LIN {X 0,Y 393.57,Z 349.625,A -85,B 0,C 180,E1 -11638.956,E2 -11638.956} C_VEL
LIN {X 0,Y 390.601,Z 337.72,A -85,B 0,C 180,E1 -11641.782,E2 -11641.782} C_VEL
LIN {X 0,Y 390.037,Z 335.528,A -85,B 0,C 180,E1 -11642.376,E2 -11642.376} C_VEL
LIN {X 0,Y 390.052,Z 335.522,A -85,B 0,C 180,E1 -11645.825,E2 -11645.825} C_VEL
LIN {X 0,Y 390.064,Z 335.516,A -85,B 0,C 180,E1 -11649.217,E2 -11649.217} C_VEL
LIN {X 0,Y 390.037,Z 335.522,A -85,B 0,C 180,E1 -11652.373,E2 -11652.373} C_VEL
LIN {X 0,Y 390.038,Z 335.516,A -85,B 0,C 180,E1 -11655.354,E2 -11655.354} C_VEL
LIN {X 0,Y 390.024,Z 335.526,A -85,B 0,C 180,E1 -11658.186,E2 -11658.186} C_VEL
LIN {X 0,Y 390.082,Z 335.519,A -85,B 0,C 180,E1 -11660.907,E2 -11660.907} C_VEL
LIN {X 0,Y 390.077,Z 335.515,A -85,B 0,C 180,E1 -11664.792,E2 -11664.792} C_VEL
LIN {X 0,Y 390.014,Z 335.517,A -85,B 0,C 180,E1 -11668.495,E2 -11668.495} C_VEL
LIN {X 0,Y 390.028,Z 335.519,A -85,B 0,C 180,E1 -11672.063,E2 -11672.063} C_VEL
LIN {X 0,Y 390.042,Z 335.52,A -85,B 0,C 180,E1 -11675.517,E2 -11675.517} C_VEL
LIN {X 0,Y 390.045,Z 335.519,A -85,B 0,C 180,E1 -11678.877,E2 -11678.877} C_VEL
LIN {X 0,Y 390.1,Z 335.516,A -85,B 0,C 180,E1 -11682.166,E2 -11682.166} C_VEL
LIN {X 0,Y 390.131,Z 335.512,A -85,B 0,C 180,E1 -11685.392,E2 -11685.392} C_VEL
LIN {X 0,Y 390.123,Z 335.505,A -85,B 0,C 180,E1 -11688.571,E2 -11688.571} C_VEL
LIN {X 0,Y 390.245,Z 335.493,A -85,B 0,C 180,E1 -11692.087,E2 -11692.087} C_VEL
LIN {X 0,Y 390.191,Z 335.503,A -85,B 0,C 180,E1 -11694.833,E2 -11694.833} C_VEL
LIN {X 0,Y 390.395,Z 335.473,A -85,B 0,C 180,E1 -11697.937,E2 -11697.937} C_VEL
LIN {X 0,Y 390.402,Z 335.471,A -85,B 0,C 180,E1 -11702.064,E2 -11702.064} C_VEL
LIN {X 0,Y 390.268,Z 335.49,A -85,B 0,C 180,E1 -11706.592,E2 -11706.592} C_VEL
LIN {X 0,Y 390.181,Z 335.51,A -85,B 0,C 180,E1 -11709.33,E2 -11709.33} C_VEL
LIN {X 0,Y 390.16,Z 335.5,A -85,B 0,C 180,E1 -11712.484,E2 -11712.484} C_VEL
LIN {X 0,Y 390.128,Z 335.508,A -85,B 0,C 180,E1 -11715.678,E2 -11715.678} C_VEL
LIN {X 0,Y 390.093,Z 335.521,A -85,B 0,C 180,E1 -11718.923,E2 -11718.923} C_VEL
LIN {X 0,Y 390.029,Z 335.524,A -85,B 0,C 180,E1 -11722.235,E2 -11722.235} C_VEL
LIN {X 0,Y 390.112,Z 335.514,A -85,B 0,C 180,E1 -11725.744,E2 -11725.744} C_VEL
LIN {X 0,Y 390.052,Z 335.525,A -85,B 0,C 180,E1 -11729.111,E2 -11729.111} C_VEL
LIN {X 0,Y 390.037,Z 335.527,A -85,B 0,C 180,E1 -11732.723,E2 -11732.723} C_VEL
LIN {X 0,Y 390.05,Z 335.521,A -85,B 0,C 180,E1 -11735.826,E2 -11735.826} C_VEL
LIN {X 0,Y 390.062,Z 335.519,A -85,B 0,C 180,E1 -11739.219,E2 -11739.219} C_VEL
LIN {X 0,Y 390.039,Z 335.524,A -85,B 0,C 180,E1 -11742.375,E2 -11742.375} C_VEL
LIN {X 0,Y 390.042,Z 335.524,A -85,B 0,C 180,E1 -11745.356,E2 -11745.356} C_VEL
LIN {X 0,Y 390.03,Z 335.529,A -85,B 0,C 180,E1 -11748.188,E2 -11748.188} C_VEL
LIN {X 0,Y 390.091,Z 335.52,A -85,B 0,C 180,E1 -11750.909,E2 -11750.909} C_VEL
LIN {X 0,Y 390.088,Z 335.514,A -85,B 0,C 180,E1 -11754.795,E2 -11754.795} C_VEL
LIN {X 0,Y 390.112,Z 335.621,A -85,B 0,C 180,E1 -11755.505,E2 -11755.505} C_VEL
LIN {X 0,Y 392.898,Z 347.642,A -85,B 0,C 180,E1 -11758.619,E2 -11758.619} C_VEL
LIN {X 0,Y 399.836,Z 363.88,A -85,B 0,C 180,E1 -11759.462,E2 -11759.462} C_VEL
LIN {X 0,Y 402.263,Z 374.857,A -85,B 0,C 180,E1 -11759.852,E2 -11759.852} C_VEL
LIN {X 0,Y 400.409,Z 475.85,A -85,B 0,C 180,E1 -11761.69,E2 -11761.69} C_VEL
LIN {X 0,Y 399.994,Z 490.23,A -85,B 0,C 180,E1 -11762.037,E2 -11762.037} C_VEL
LIN {X 0,Y 399.273,Z 503.733,A -85,B 0,C 180,E1 -11762.552,E2 -11762.552} C_VEL
LIN {X 0,Y 398.397,Z 517.078,A -85,B 0,C 180,E1 -11763.268,E2 -11763.268} C_VEL
LIN {X 0,Y 397.243,Z 529.931,A -85,B 0,C 180,E1 -11764.162,E2 -11764.162} C_VEL
LIN {X 0,Y 395.992,Z 541.893,A -85,B 0,C 180,E1 -11765.211,E2 -11765.211} C_VEL
LIN {X 0,Y 394.754,Z 552.816,A -85,B 0,C 180,E1 -11766.386,E2 -11766.386} C_VEL
LIN {X 0,Y 393.58,Z 562.901,A -85,B 0,C 180,E1 -11767.701,E2 -11767.701} C_VEL
LIN {X 0,Y 392.438,Z 572.905,A -85,B 0,C 180,E1 -11769.287,E2 -11769.287} C_VEL
LIN {X 0,Y 391.363,Z 581.167,A -85,B 0,C 180,E1 -11770.87,E2 -11770.87} C_VEL
LIN {X 0,Y 390.513,Z 588.281,A -85,B 0,C 180,E1 -11772.524,E2 -11772.524} C_VEL
LIN {X 0,Y 389.805,Z 594.521,A -85,B 0,C 180,E1 -11774.31,E2 -11774.31} C_VEL
LIN {X 0,Y 389.248,Z 600.25,A -85,B 0,C 180,E1 -11776.425,E2 -11776.425} C_VEL
LIN {X 0,Y 388.893,Z 604.387,A -85,B 0,C 180,E1 -11778.534,E2 -11778.534} C_VEL
LIN {X 0,Y 388.65,Z 607.065,A -85,B 0,C 180,E1 -11780.634,E2 -11780.634} C_VEL
LIN {X 0,Y 388.664,Z 608.364,A -85,B 0,C 180,E1 -11782.728,E2 -11782.728} C_VEL
LIN {X 0,Y 388.733,Z 608.487,A -85,B 0,C 180,E1 -11783.917,E2 -11783.917} C_VEL
LIN {X 0,Y 388.682,Z 607.807,A -85,B 0,C 180,E1 -11785.852,E2 -11785.852} C_VEL
LIN {X 0,Y 388.764,Z 605.775,A -85,B 0,C 180,E1 -11787.928,E2 -11787.928} C_VEL
LIN {X 0,Y 388.858,Z 602.376,A -85,B 0,C 180,E1 -11790,E2 -11790} C_VEL
LIN {X 0,Y 389.112,Z 597.509,A -85,B 0,C 180,E1 -11792.07,E2 -11792.07} C_VEL
LIN {X 0,Y 389.319,Z 595.751,A -85,B 0,C 180,E1 -11792.69,E2 -11792.69} C_VEL
LIN {X 0,Y 388.781,Z 593.369,A -85,B 0,C 180,E1 -11793.478,E2 -11793.478} C_VEL
LIN {X 0,Y 386.379,Z 589.112,A -85,B 0,C 180,E1 -11794.754,E2 -11794.754} C_VEL
LIN {X 0,Y 384.109,Z 584.4,A -85,B 0,C 180,E1 -11796.006,E2 -11796.006} C_VEL
LIN {X 0,Y 383.785,Z 581.149,A -85,B 0,C 180,E1 -11796.744,E2 -11796.744} C_VEL
LIN {X 0,Y 384.777,Z 572.525,A -85,B 0,C 180,E1 -11798.402,E2 -11798.402} C_VEL
LIN {X 0,Y 385.604,Z 563.561,A -85,B 0,C 180,E1 -11799.838,E2 -11799.838} C_VEL
LIN {X 0,Y 386.684,Z 552.994,A -85,B 0,C 180,E1 -11801.24,E2 -11801.24} C_VEL
LIN {X 0,Y 387.949,Z 540.823,A -85,B 0,C 180,E1 -11802.555,E2 -11802.555} C_VEL
LIN {X 0,Y 388.984,Z 529.039,A -85,B 0,C 180,E1 -11803.584,E2 -11803.584} C_VEL
LIN {X 0,Y 389.979,Z 516.108,A -85,B 0,C 180,E1 -11804.48,E2 -11804.48} C_VEL
LIN {X 0,Y 390.819,Z 502.017,A -85,B 0,C 180,E1 -11805.214,E2 -11805.214} C_VEL
LIN {X 0,Y 391.478,Z 488.049,A -85,B 0,C 180,E1 -11805.722,E2 -11805.722} C_VEL
LIN {X 0,Y 391.849,Z 470.558,A -85,B 0,C 180,E1 -11806.107,E2 -11806.107} C_VEL
LIN {X 0,Y 393.349,Z 374.86,A -85,B 0,C 180,E1 -11807.863,E2 -11807.863} C_VEL
LIN {X 0,Y 390.127,Z 359.978,A -85,B 0,C 180,E1 -11808.344,E2 -11808.344} C_VEL
LIN {X 0,Y 385.42,Z 347.358,A -85,B 0,C 180,E1 -11808.914,E2 -11808.914} C_VEL
LIN {X 0,Y 383.01,Z 336.403,A -85,B 0,C 180,E1 -11811.671,E2 -11811.671} C_VEL
LIN {X 0,Y 383.054,Z 336.395,A -85,B 0,C 180,E1 -11814.959,E2 -11814.959} C_VEL
LIN {X 0,Y 383.031,Z 336.394,A -85,B 0,C 180,E1 -11818.269,E2 -11818.269} C_VEL
LIN {X 0,Y 383.01,Z 336.4,A -85,B 0,C 180,E1 -11822.149,E2 -11822.149} C_VEL
LIN {X 0,Y 383.018,Z 336.396,A -85,B 0,C 180,E1 -11824.667,E2 -11824.667} C_VEL
LIN {X 0,Y 383.001,Z 336.402,A -85,B 0,C 180,E1 -11827.903,E2 -11827.903} C_VEL
LIN {X 0,Y 382.982,Z 336.393,A -85,B 0,C 180,E1 -11831.346,E2 -11831.346} C_VEL
LIN {X 0,Y 382.993,Z 336.398,A -85,B 0,C 180,E1 -11834.302,E2 -11834.302} C_VEL
LIN {X 0,Y 383.007,Z 336.403,A -85,B 0,C 180,E1 -11837.239,E2 -11837.239} C_VEL
LIN {X 0,Y 383.009,Z 336.398,A -85,B 0,C 180,E1 -11840.413,E2 -11840.413} C_VEL
LIN {X 0,Y 383.019,Z 336.397,A -85,B 0,C 180,E1 -11844.043,E2 -11844.043} C_VEL
LIN {X 0,Y 382.98,Z 336.403,A -85,B 0,C 180,E1 -11847.577,E2 -11847.577} C_VEL
LIN {X 0,Y 382.985,Z 336.4,A -85,B 0,C 180,E1 -11850.299,E2 -11850.299} C_VEL
LIN {X 0,Y 383.062,Z 336.387,A -85,B 0,C 180,E1 -11854.023,E2 -11854.023} C_VEL
LIN {X 0,Y 382.982,Z 336.4,A -85,B 0,C 180,E1 -11857.333,E2 -11857.333} C_VEL
LIN {X 0,Y 383.049,Z 336.383,A -85,B 0,C 180,E1 -11860.715,E2 -11860.715} C_VEL
LIN {X 0,Y 383.07,Z 336.39,A -85,B 0,C 180,E1 -11864.026,E2 -11864.026} C_VEL
LIN {X 0,Y 383.125,Z 336.369,A -85,B 0,C 180,E1 -11867.283,E2 -11867.283} C_VEL
LIN {X 0,Y 383.131,Z 336.383,A -85,B 0,C 180,E1 -11870.497,E2 -11870.497} C_VEL
LIN {X 0,Y 383.248,Z 336.362,A -85,B 0,C 180,E1 -11873.683,E2 -11873.683} C_VEL
LIN {X 0,Y 383.364,Z 336.35,A -85,B 0,C 180,E1 -11877.898,E2 -11877.898} C_VEL
LIN {X 0,Y 383.355,Z 336.353,A -85,B 0,C 180,E1 -11882.101,E2 -11882.101} C_VEL
LIN {X 0,Y 383.221,Z 336.376,A -85,B 0,C 180,E1 -11886.317,E2 -11886.317} C_VEL
LIN {X 0,Y 383.128,Z 336.373,A -85,B 0,C 180,E1 -11889.502,E2 -11889.502} C_VEL
LIN {X 0,Y 383.115,Z 336.385,A -85,B 0,C 180,E1 -11893.536,E2 -11893.536} C_VEL
LIN {X 0,Y 383.083,Z 336.386,A -85,B 0,C 180,E1 -11897.069,E2 -11897.069} C_VEL
LIN {X 0,Y 383.018,Z 336.388,A -85,B 0,C 180,E1 -11900.647,E2 -11900.647} C_VEL
LIN {X 0,Y 383.007,Z 336.4,A -85,B 0,C 180,E1 -11903.809,E2 -11903.809} C_VEL
LIN {X 0,Y 382.984,Z 336.398,A -85,B 0,C 180,E1 -11907.307,E2 -11907.307} C_VEL
LIN {X 0,Y 382.973,Z 336.399,A -85,B 0,C 180,E1 -11910.919,E2 -11910.919} C_VEL
LIN {X 0,Y 383.01,Z 336.397,A -85,B 0,C 180,E1 -11914.669,E2 -11914.669} C_VEL
LIN {X 0,Y 382.992,Z 336.403,A -85,B 0,C 180,E1 -11917.904,E2 -11917.904} C_VEL
LIN {X 0,Y 382.977,Z 336.395,A -85,B 0,C 180,E1 -11921.348,E2 -11921.348} C_VEL
LIN {X 0,Y 382.989,Z 336.401,A -85,B 0,C 180,E1 -11924.304,E2 -11924.304} C_VEL
LIN {X 0,Y 383.004,Z 336.401,A -85,B 0,C 180,E1 -11927.241,E2 -11927.241} C_VEL
LIN {X 0,Y 383.008,Z 336.403,A -85,B 0,C 180,E1 -11930.415,E2 -11930.415} C_VEL
LIN {X 0,Y 383.021,Z 336.404,A -85,B 0,C 180,E1 -11934.045,E2 -11934.045} C_VEL
LIN {X 0,Y 382.983,Z 336.407,A -85,B 0,C 180,E1 -11937.579,E2 -11937.579} C_VEL
LIN {X 0,Y 383.029,Z 336.457,A -85,B 0,C 180,E1 -11938.703,E2 -11938.703} C_VEL
LIN {X 0,Y 386.124,Z 349.978,A -85,B 0,C 180,E1 -11941.756,E2 -11941.756} C_VEL
LIN {X 0,Y 387.81,Z 358.69,A -85,B 0,C 180,E1 -11943.642,E2 -11943.642} C_VEL
LIN {X 0,Y 387.16,Z 366.783,A -85,B 0,C 180,E1 -11945.234,E2 -11945.234} C_VEL
LIN {X 0,Y 393.011,Z 400.789,A -85,B 0,C 180,E1 -11946.256,E2 -11946.256} C_VEL
LIN {X 0,Y 391.334,Z 503.62,A -85,B 0,C 180,E1 -11948.156,E2 -11948.156} C_VEL
LIN {X 0,Y 390.713,Z 518.128,A -85,B 0,C 180,E1 -11948.605,E2 -11948.605} C_VEL
LIN {X 0,Y 389.861,Z 531.407,A -85,B 0,C 180,E1 -11949.213,E2 -11949.213} C_VEL
LIN {X 0,Y 388.924,Z 544.111,A -85,B 0,C 180,E1 -11949.994,E2 -11949.994} C_VEL
LIN {X 0,Y 387.84,Z 556.483,A -85,B 0,C 180,E1 -11950.964,E2 -11950.964} C_VEL
LIN {X 0,Y 386.582,Z 568.511,A -85,B 0,C 180,E1 -11952.135,E2 -11952.135} C_VEL
LIN {X 0,Y 385.57,Z 578.507,A -85,B 0,C 180,E1 -11953.317,E2 -11953.317} C_VEL
LIN {X 0,Y 384.404,Z 589.507,A -85,B 0,C 180,E1 -11954.899,E2 -11954.899} C_VEL
LIN {X 0,Y 383.61,Z 598.593,A -85,B 0,C 180,E1 -11956.492,E2 -11956.492} C_VEL
LIN {X 0,Y 382.793,Z 607.273,A -85,B 0,C 180,E1 -11958.349,E2 -11958.349} C_VEL
LIN {X 0,Y 382.221,Z 613.351,A -85,B 0,C 180,E1 -11959.94,E2 -11959.94} C_VEL
LIN {X 0,Y 381.84,Z 619.821,A -85,B 0,C 180,E1 -11962.066,E2 -11962.066} C_VEL
LIN {X 0,Y 381.695,Z 623.987,A -85,B 0,C 180,E1 -11963.869,E2 -11963.869} C_VEL
LIN {X 0,Y 381.612,Z 627.209,A -85,B 0,C 180,E1 -11965.776,E2 -11965.776} C_VEL
LIN {X 0,Y 381.572,Z 629.444,A -85,B 0,C 180,E1 -11967.889,E2 -11967.889} C_VEL
LIN {X 0,Y 381.637,Z 630.326,A -85,B 0,C 180,E1 -11970,E2 -11970} C_VEL
LIN {X 0,Y 381.556,Z 629.867,A -85,B 0,C 180,E1 -11972.111,E2 -11972.111} C_VEL
LIN {X 0,Y 381.608,Z 628.078,A -85,B 0,C 180,E1 -11974.225,E2 -11974.225} C_VEL
LIN {X 0,Y 381.709,Z 624.917,A -85,B 0,C 180,E1 -11976.342,E2 -11976.342} C_VEL
LIN {X 0,Y 381.975,Z 620.277,A -85,B 0,C 180,E1 -11978.464,E2 -11978.464} C_VEL
LIN {X 0,Y 382.462,Z 614.001,A -85,B 0,C 180,E1 -11980.588,E2 -11980.588} C_VEL
LIN {X 0,Y 383.328,Z 607.034,A -85,B 0,C 180,E1 -11982.44,E2 -11982.44} C_VEL
LIN {X 0,Y 384.244,Z 598.326,A -85,B 0,C 180,E1 -11984.313,E2 -11984.313} C_VEL
LIN {X 0,Y 385.352,Z 589.431,A -85,B 0,C 180,E1 -11985.876,E2 -11985.876} C_VEL
LIN {X 0,Y 386.714,Z 578.573,A -85,B 0,C 180,E1 -11987.449,E2 -11987.449} C_VEL
LIN {X 0,Y 388.137,Z 567.574,A -85,B 0,C 180,E1 -11988.747,E2 -11988.747} C_VEL
LIN {X 0,Y 389.527,Z 555.52,A -85,B 0,C 180,E1 -11989.91,E2 -11989.91} C_VEL
LIN {X 0,Y 390.77,Z 543.255,A -85,B 0,C 180,E1 -11990.858,E2 -11990.858} C_VEL
LIN {X 0,Y 391.844,Z 530.301,A -85,B 0,C 180,E1 -11991.641,E2 -11991.641} C_VEL
LIN {X 0,Y 392.871,Z 515.89,A -85,B 0,C 180,E1 -11992.272,E2 -11992.272} C_VEL
LIN {X 0,Y 393.576,Z 501.721,A -85,B 0,C 180,E1 -11992.68,E2 -11992.68} C_VEL
LIN {X 0,Y 395.527,Z 402.682,A -85,B 0,C 180,E1 -11994.519,E2 -11994.519} C_VEL
LIN {X 0,Y 393.52,Z 390.342,A -85,B 0,C 180,E1 -11994.912,E2 -11994.912} C_VEL
LIN {X 0,Y 388.517,Z 366.499,A -85,B 0,C 180,E1 -11995.802,E2 -11995.802} C_VEL
LIN {X 0,Y 388.923,Z 362.7,A -85,B 0,C 180,E1 -11996.566,E2 -11996.566} C_VEL
LIN {X 0,Y 387.175,Z 353.233,A -85,B 0,C 180,E1 -11998.71,E2 -11998.71} C_VEL
LIN {X 0,Y 384.094,Z 340.649,A -85,B 0,C 180,E1 -12001.738,E2 -12001.738} C_VEL
LIN {X 0,Y 382.991,Z 336.405,A -85,B 0,C 180,E1 -12002.83,E2 -12002.83} C_VEL
LIN {X 0,Y 383.028,Z 336.397,A -85,B 0,C 180,E1 -12006.164,E2 -12006.164} C_VEL
LIN {X 0,Y 383.003,Z 336.389,A -85,B 0,C 180,E1 -12009.958,E2 -12009.958} C_VEL
LIN {X 0,Y 383,Z 336.395,A -85,B 0,C 180,E1 -12012.778,E2 -12012.778} C_VEL
LIN {X 0,Y 382.991,Z 336.397,A -85,B 0,C 180,E1 -12015.788,E2 -12015.788} C_VEL
LIN {X 0,Y 382.981,Z 336.402,A -85,B 0,C 180,E1 -12018.795,E2 -12018.795} C_VEL
LIN {X 0,Y 382.992,Z 336.402,A -85,B 0,C 180,E1 -12022.096,E2 -12022.096} C_VEL
LIN {X 0,Y 383.01,Z 336.395,A -85,B 0,C 180,E1 -12025.331,E2 -12025.331} C_VEL
LIN {X 0,Y 382.973,Z 336.39,A -85,B 0,C 180,E1 -12029.081,E2 -12029.081} C_VEL
LIN {X 0,Y 382.984,Z 336.401,A -85,B 0,C 180,E1 -12032.693,E2 -12032.693} C_VEL
LIN {X 0,Y 383.004,Z 336.399,A -85,B 0,C 180,E1 -12036.191,E2 -12036.191} C_VEL
LIN {X 0,Y 383.045,Z 336.391,A -85,B 0,C 180,E1 -12039.598,E2 -12039.598} C_VEL
LIN {X 0,Y 383.083,Z 336.388,A -85,B 0,C 180,E1 -12042.931,E2 -12042.931} C_VEL
LIN {X 0,Y 383.115,Z 336.385,A -85,B 0,C 180,E1 -12046.464,E2 -12046.464} C_VEL
LIN {X 0,Y 383.123,Z 336.384,A -85,B 0,C 180,E1 -12050.498,E2 -12050.498} C_VEL
LIN {X 0,Y 383.228,Z 336.369,A -85,B 0,C 180,E1 -12053.683,E2 -12053.683} C_VEL
LIN {X 0,Y 383.361,Z 336.349,A -85,B 0,C 180,E1 -12057.899,E2 -12057.899} C_VEL
LIN {X 0,Y 383.368,Z 336.347,A -85,B 0,C 180,E1 -12062.102,E2 -12062.102} C_VEL
LIN {X 0,Y 383.229,Z 336.367,A -85,B 0,C 180,E1 -12066.582,E2 -12066.582} C_VEL
LIN {X 0,Y 383.132,Z 336.386,A -85,B 0,C 180,E1 -12069.503,E2 -12069.503} C_VEL
LIN {X 0,Y 383.116,Z 336.387,A -85,B 0,C 180,E1 -12073.537,E2 -12073.537} C_VEL
LIN {X 0,Y 383.085,Z 336.387,A -85,B 0,C 180,E1 -12077.07,E2 -12077.07} C_VEL
LIN {X 0,Y 383.02,Z 336.395,A -85,B 0,C 180,E1 -12080.648,E2 -12080.648} C_VEL
LIN {X 0,Y 383.018,Z 336.395,A -85,B 0,C 180,E1 -12083.809,E2 -12083.809} C_VEL
LIN {X 0,Y 383.073,Z 336.391,A -85,B 0,C 180,E1 -12086.124,E2 -12086.124} C_VEL
LIN {X 0,Y 382.985,Z 336.402,A -85,B 0,C 180,E1 -12089.701,E2 -12089.701} C_VEL
LIN {X 0,Y 382.997,Z 336.399,A -85,B 0,C 180,E1 -12093.402,E2 -12093.402} C_VEL
LIN {X 0,Y 383.026,Z 336.398,A -85,B 0,C 180,E1 -12096.166,E2 -12096.166} C_VEL
LIN {X 0,Y 383.004,Z 336.398,A -85,B 0,C 180,E1 -12099.96,E2 -12099.96} C_VEL
LIN {X 0,Y 383.002,Z 336.401,A -85,B 0,C 180,E1 -12102.78,E2 -12102.78} C_VEL
LIN {X 0,Y 382.994,Z 336.403,A -85,B 0,C 180,E1 -12105.79,E2 -12105.79} C_VEL
LIN {X 0,Y 382.987,Z 336.404,A -85,B 0,C 180,E1 -12108.797,E2 -12108.797} C_VEL
LIN {X 0,Y 383.001,Z 336.402,A -85,B 0,C 180,E1 -12112.097,E2 -12112.097} C_VEL
LIN {X 0,Y 383.043,Z 336.405,A -85,B 0,C 180,E1 -12115.016,E2 -12115.016} C_VEL
LIN {X 0,Y 385.732,Z 347.824,A -85,B 0,C 180,E1 -12118.06,E2 -12118.06} C_VEL
LIN {X 0,Y 393.768,Z 366.34,A -85,B 0,C 180,E1 -12119.063,E2 -12119.063} C_VEL
LIN {X 0,Y 395.985,Z 376.393,A -85,B 0,C 180,E1 -12119.429,E2 -12119.429} C_VEL
LIN {X 0,Y 393.713,Z 484.435,A -85,B 0,C 180,E1 -12121.442,E2 -12121.442} C_VEL
LIN {X 0,Y 393.072,Z 499.2,A -85,B 0,C 180,E1 -12121.937,E2 -12121.937} C_VEL
LIN {X 0,Y 392.203,Z 512.691,A -85,B 0,C 180,E1 -12122.594,E2 -12122.594} C_VEL
LIN {X 0,Y 391.032,Z 526.043,A -85,B 0,C 180,E1 -12123.459,E2 -12123.459} C_VEL
LIN {X 0,Y 389.748,Z 539.019,A -85,B 0,C 180,E1 -12124.543,E2 -12124.543} C_VEL
LIN {X 0,Y 388.525,Z 548.942,A -85,B 0,C 180,E1 -12125.558,E2 -12125.558} C_VEL
LIN {X 0,Y 387.327,Z 558.73,A -85,B 0,C 180,E1 -12126.756,E2 -12126.756} C_VEL
LIN {X 0,Y 386.144,Z 569.091,A -85,B 0,C 180,E1 -12128.297,E2 -12128.297} C_VEL
LIN {X 0,Y 384.863,Z 578.419,A -85,B 0,C 180,E1 -12129.978,E2 -12129.978} C_VEL
LIN {X 0,Y 383.95,Z 585.772,A -85,B 0,C 180,E1 -12131.594,E2 -12131.594} C_VEL
LIN {X 0,Y 383.088,Z 592.773,A -85,B 0,C 180,E1 -12133.48,E2 -12133.48} C_VEL
LIN {X 0,Y 382.497,Z 597.598,A -85,B 0,C 180,E1 -12135.094,E2 -12135.094} C_VEL
LIN {X 0,Y 382.041,Z 602.562,A -85,B 0,C 180,E1 -12137.247,E2 -12137.247} C_VEL
LIN {X 0,Y 381.673,Z 606.003,A -85,B 0,C 180,E1 -12139.389,E2 -12139.389} C_VEL
LIN {X 0,Y 381.575,Z 608.032,A -85,B 0,C 180,E1 -12141.527,E2 -12141.527} C_VEL
LIN {X 0,Y 381.618,Z 608.712,A -85,B 0,C 180,E1 -12143.656,E2 -12143.656} C_VEL
LIN {X 0,Y 381.605,Z 608.062,A -85,B 0,C 180,E1 -12145.775,E2 -12145.775} C_VEL
LIN {X 0,Y 381.661,Z 606.078,A -85,B 0,C 180,E1 -12147.889,E2 -12147.889} C_VEL
LIN {X 0,Y 381.781,Z 602.725,A -85,B 0,C 180,E1 -12150,E2 -12150} C_VEL
LIN {X 0,Y 382.041,Z 597.908,A -85,B 0,C 180,E1 -12152.108,E2 -12152.108} C_VEL
LIN {X 0,Y 382.602,Z 591.47,A -85,B 0,C 180,E1 -12154.214,E2 -12154.214} C_VEL
LIN {X 0,Y 383.436,Z 584.305,A -85,B 0,C 180,E1 -12156.05,E2 -12156.05} C_VEL
LIN {X 0,Y 383.785,Z 581.149,A -85,B 0,C 180,E1 -12156.744,E2 -12156.744} C_VEL
LIN {X 0,Y 383.457,Z 577.764,A -85,B 0,C 180,E1 -12157.468,E2 -12157.468} C_VEL
LIN {X 0,Y 381.252,Z 572.035,A -85,B 0,C 180,E1 -12158.638,E2 -12158.638} C_VEL
LIN {X 0,Y 379.138,Z 565.824,A -85,B 0,C 180,E1 -12159.76,E2 -12159.76} C_VEL
LIN {X 0,Y 378.946,Z 561.686,A -85,B 0,C 180,E1 -12160.398,E2 -12160.398} C_VEL
LIN {X 0,Y 380.066,Z 551.42,A -85,B 0,C 180,E1 -12161.736,E2 -12161.736} C_VEL
LIN {X 0,Y 381.36,Z 539.016,A -85,B 0,C 180,E1 -12163.047,E2 -12163.047} C_VEL
LIN {X 0,Y 382.459,Z 526.738,A -85,B 0,C 180,E1 -12164.092,E2 -12164.092} C_VEL
LIN {X 0,Y 383.425,Z 514.171,A -85,B 0,C 180,E1 -12164.937,E2 -12164.937} C_VEL
LIN {X 0,Y 384.294,Z 500.068,A -85,B 0,C 180,E1 -12165.649,E2 -12165.649} C_VEL
LIN {X 0,Y 384.869,Z 486.189,A -85,B 0,C 180,E1 -12166.135,E2 -12166.135} C_VEL
LIN {X 0,Y 385.386,Z 460.471,A -85,B 0,C 180,E1 -12166.657,E2 -12166.657} C_VEL
LIN {X 0,Y 386.806,Z 376.176,A -85,B 0,C 180,E1 -12168.227,E2 -12168.227} C_VEL
LIN {X 0,Y 383.883,Z 362.519,A -85,B 0,C 180,E1 -12168.677,E2 -12168.677} C_VEL
LIN {X 0,Y 378.268,Z 347.659,A -85,B 0,C 180,E1 -12169.345,E2 -12169.345} C_VEL
LIN {X 0,Y 375.965,Z 337.282,A -85,B 0,C 180,E1 -12172.026,E2 -12172.026} C_VEL
LIN {X 0,Y 376.008,Z 337.275,A -85,B 0,C 180,E1 -12175.46,E2 -12175.46} C_VEL
LIN {X 0,Y 375.962,Z 337.273,A -85,B 0,C 180,E1 -12179.079,E2 -12179.079} C_VEL
LIN {X 0,Y 375.95,Z 337.277,A -85,B 0,C 180,E1 -12182.827,E2 -12182.827} C_VEL
LIN {X 0,Y 375.958,Z 337.272,A -85,B 0,C 180,E1 -12185.414,E2 -12185.414} C_VEL
LIN {X 0,Y 375.975,Z 337.275,A -85,B 0,C 180,E1 -12188.27,E2 -12188.27} C_VEL
LIN {X 0,Y 375.932,Z 337.275,A -85,B 0,C 180,E1 -12191.599,E2 -12191.599} C_VEL
LIN {X 0,Y 375.924,Z 337.281,A -85,B 0,C 180,E1 -12195.267,E2 -12195.267} C_VEL
LIN {X 0,Y 375.93,Z 337.275,A -85,B 0,C 180,E1 -12198.398,E2 -12198.398} C_VEL
LIN {X 0,Y 375.967,Z 337.272,A -85,B 0,C 180,E1 -12201.729,E2 -12201.729} C_VEL
LIN {X 0,Y 375.974,Z 337.276,A -85,B 0,C 180,E1 -12205.332,E2 -12205.332} C_VEL
LIN {X 0,Y 375.951,Z 337.277,A -85,B 0,C 180,E1 -12208.437,E2 -12208.437} C_VEL
LIN {X 0,Y 375.975,Z 337.263,A -85,B 0,C 180,E1 -12212.139,E2 -12212.139} C_VEL
LIN {X 0,Y 375.983,Z 337.27,A -85,B 0,C 180,E1 -12214.537,E2 -12214.537} C_VEL
LIN {X 0,Y 375.947,Z 337.273,A -85,B 0,C 180,E1 -12218.044,E2 -12218.044} C_VEL
LIN {X 0,Y 375.993,Z 337.27,A -85,B 0,C 180,E1 -12221.472,E2 -12221.472} C_VEL
LIN {X 0,Y 376.048,Z 337.265,A -85,B 0,C 180,E1 -12224.832,E2 -12224.832} C_VEL
LIN {X 0,Y 376.036,Z 337.252,A -85,B 0,C 180,E1 -12228.136,E2 -12228.136} C_VEL
LIN {X 0,Y 376.189,Z 337.247,A -85,B 0,C 180,E1 -12231.941,E2 -12231.941} C_VEL
LIN {X 0,Y 376.145,Z 337.24,A -85,B 0,C 180,E1 -12234.639,E2 -12234.639} C_VEL
LIN {X 0,Y 376.33,Z 337.226,A -85,B 0,C 180,E1 -12237.859,E2 -12237.859} C_VEL
LIN {X 0,Y 376.319,Z 337.229,A -85,B 0,C 180,E1 -12242.14,E2 -12242.14} C_VEL
LIN {X 0,Y 376.181,Z 337.254,A -85,B 0,C 180,E1 -12246.436,E2 -12246.436} C_VEL
LIN {X 0,Y 376.099,Z 337.249,A -85,B 0,C 180,E1 -12249.682,E2 -12249.682} C_VEL
LIN {X 0,Y 376.079,Z 337.262,A -85,B 0,C 180,E1 -12253.657,E2 -12253.657} C_VEL
LIN {X 0,Y 376.022,Z 337.266,A -85,B 0,C 180,E1 -12257.4,E2 -12257.4} C_VEL
LIN {X 0,Y 375.969,Z 337.265,A -85,B 0,C 180,E1 -12260.832,E2 -12260.832} C_VEL
LIN {X 0,Y 375.967,Z 337.276,A -85,B 0,C 180,E1 -12264.283,E2 -12264.283} C_VEL
LIN {X 0,Y 375.925,Z 337.282,A -85,B 0,C 180,E1 -12267.864,E2 -12267.864} C_VEL
LIN {X 0,Y 375.948,Z 337.277,A -85,B 0,C 180,E1 -12271.563,E2 -12271.563} C_VEL
LIN {X 0,Y 375.949,Z 337.278,A -85,B 0,C 180,E1 -12275.416,E2 -12275.416} C_VEL
LIN {X 0,Y 375.967,Z 337.278,A -85,B 0,C 180,E1 -12278.271,E2 -12278.271} C_VEL
LIN {X 0,Y 375.927,Z 337.272,A -85,B 0,C 180,E1 -12281.601,E2 -12281.601} C_VEL
LIN {X 0,Y 375.921,Z 337.282,A -85,B 0,C 180,E1 -12285.269,E2 -12285.269} C_VEL
LIN {X 0,Y 375.928,Z 337.282,A -85,B 0,C 180,E1 -12288.4,E2 -12288.4} C_VEL
LIN {X 0,Y 375.968,Z 337.283,A -85,B 0,C 180,E1 -12291.731,E2 -12291.731} C_VEL
LIN {X 0,Y 375.976,Z 337.282,A -85,B 0,C 180,E1 -12295.333,E2 -12295.333} C_VEL
LIN {X 0,Y 375.986,Z 337.443,A -85,B 0,C 180,E1 -12298.363,E2 -12298.363} C_VEL
LIN {X 0,Y 378.799,Z 349.513,A -85,B 0,C 180,E1 -12301.16,E2 -12301.16} C_VEL
LIN {X 0,Y 380.817,Z 359.685,A -85,B 0,C 180,E1 -12303.415,E2 -12303.415} C_VEL
LIN {X 0,Y 380.598,Z 364.25,A -85,B 0,C 180,E1 -12304.341,E2 -12304.341} C_VEL
LIN {X 0,Y 380.355,Z 366.638,A -85,B 0,C 180,E1 -12304.817,E2 -12304.817} C_VEL
LIN {X 0,Y 386.433,Z 401.807,A -85,B 0,C 180,E1 -12305.893,E2 -12305.893} C_VEL
LIN {X 0,Y 384.643,Z 504.571,A -85,B 0,C 180,E1 -12307.827,E2 -12307.827} C_VEL
LIN {X 0,Y 383.956,Z 518.558,A -85,B 0,C 180,E1 -12308.28,E2 -12308.28} C_VEL
LIN {X 0,Y 383.107,Z 531.674,A -85,B 0,C 180,E1 -12308.899,E2 -12308.899} C_VEL
LIN {X 0,Y 382.063,Z 544.932,A -85,B 0,C 180,E1 -12309.741,E2 -12309.741} C_VEL
LIN {X 0,Y 380.921,Z 557.295,A -85,B 0,C 180,E1 -12310.744,E2 -12310.744} C_VEL
LIN {X 0,Y 379.638,Z 569.147,A -85,B 0,C 180,E1 -12311.936,E2 -12311.936} C_VEL
LIN {X 0,Y 378.466,Z 579.986,A -85,B 0,C 180,E1 -12313.272,E2 -12313.272} C_VEL
LIN {X 0,Y 377.317,Z 590.711,A -85,B 0,C 180,E1 -12314.885,E2 -12314.885} C_VEL
LIN {X 0,Y 376.518,Z 599.742,A -85,B 0,C 180,E1 -12316.543,E2 -12316.543} C_VEL
LIN {X 0,Y 375.694,Z 608.038,A -85,B 0,C 180,E1 -12318.399,E2 -12318.399} C_VEL
LIN {X 0,Y 375.06,Z 614.844,A -85,B 0,C 180,E1 -12320.291,E2 -12320.291} C_VEL
LIN {X 0,Y 374.728,Z 620.88,A -85,B 0,C 180,E1 -12322.456,E2 -12322.456} C_VEL
LIN {X 0,Y 374.546,Z 625.301,A -85,B 0,C 180,E1 -12324.617,E2 -12324.617} C_VEL
LIN {X 0,Y 374.539,Z 626.957,A -85,B 0,C 180,E1 -12325.696,E2 -12325.696} C_VEL
LIN {X 0,Y 374.471,Z 629.214,A -85,B 0,C 180,E1 -12327.849,E2 -12327.849} C_VEL
LIN {X 0,Y 374.552,Z 630.119,A -85,B 0,C 180,E1 -12330,E2 -12330} C_VEL
LIN {X 0,Y 374.455,Z 629.682,A -85,B 0,C 180,E1 -12332.151,E2 -12332.151} C_VEL
LIN {X 0,Y 374.512,Z 627.915,A -85,B 0,C 180,E1 -12334.305,E2 -12334.305} C_VEL
LIN {X 0,Y 374.629,Z 624.777,A -85,B 0,C 180,E1 -12336.463,E2 -12336.463} C_VEL
LIN {X 0,Y 374.93,Z 620.173,A -85,B 0,C 180,E1 -12338.624,E2 -12338.624} C_VEL
LIN {X 0,Y 375.437,Z 613.928,A -85,B 0,C 180,E1 -12340.789,E2 -12340.789} C_VEL
LIN {X 0,Y 376.357,Z 606.993,A -85,B 0,C 180,E1 -12342.674,E2 -12342.674} C_VEL
LIN {X 0,Y 377.283,Z 598.648,A -85,B 0,C 180,E1 -12344.516,E2 -12344.516} C_VEL
LIN {X 0,Y 378.489,Z 589.467,A -85,B 0,C 180,E1 -12346.172,E2 -12346.172} C_VEL
LIN {X 0,Y 379.672,Z 580.605,A -85,B 0,C 180,E1 -12347.505,E2 -12347.505} C_VEL
LIN {X 0,Y 381.273,Z 568.887,A -85,B 0,C 180,E1 -12348.958,E2 -12348.958} C_VEL
LIN {X 0,Y 382.721,Z 557.166,A -85,B 0,C 180,E1 -12350.139,E2 -12350.139} C_VEL
LIN {X 0,Y 383.947,Z 545.735,A -85,B 0,C 180,E1 -12351.075,E2 -12351.075} C_VEL
LIN {X 0,Y 385.029,Z 533.076,A -85,B 0,C 180,E1 -12351.903,E2 -12351.903} C_VEL
LIN {X 0,Y 386.18,Z 519.168,A -85,B 0,C 180,E1 -12352.574,E2 -12352.574} C_VEL
LIN {X 0,Y 387.044,Z 504.642,A -85,B 0,C 180,E1 -12353.049,E2 -12353.049} C_VEL
LIN {X 0,Y 389.134,Z 402.526,A -85,B 0,C 180,E1 -12354.992,E2 -12354.992} C_VEL
LIN {X 0,Y 384.906,Z 380.23,A -85,B 0,C 180,E1 -12355.773,E2 -12355.773} C_VEL
LIN {X 0,Y 381.872,Z 366.336,A -85,B 0,C 180,E1 -12356.322,E2 -12356.322} C_VEL
LIN {X 0,Y 382.09,Z 364.093,A -85,B 0,C 180,E1 -12356.784,E2 -12356.784} C_VEL
LIN {X 0,Y 380.25,Z 354.526,A -85,B 0,C 180,E1 -12359.007,E2 -12359.007} C_VEL
LIN {X 0,Y 377.154,Z 342.074,A -85,B 0,C 180,E1 -12362.077,E2 -12362.077} C_VEL
LIN {X 0,Y 375.965,Z 337.281,A -85,B 0,C 180,E1 -12363.304,E2 -12363.304} C_VEL
LIN {X 0,Y 375.949,Z 337.271,A -85,B 0,C 180,E1 -12366.74,E2 -12366.74} C_VEL
LIN {X 0,Y 375.983,Z 337.263,A -85,B 0,C 180,E1 -12369.97,E2 -12369.97} C_VEL
LIN {X 0,Y 375.924,Z 337.277,A -85,B 0,C 180,E1 -12373.765,E2 -12373.765} C_VEL
LIN {X 0,Y 375.928,Z 337.278,A -85,B 0,C 180,E1 -12376.81,E2 -12376.81} C_VEL
LIN {X 0,Y 375.955,Z 337.281,A -85,B 0,C 180,E1 -12380.537,E2 -12380.537} C_VEL
LIN {X 0,Y 375.956,Z 337.278,A -85,B 0,C 180,E1 -12383.495,E2 -12383.495} C_VEL
LIN {X 0,Y 375.952,Z 337.277,A -85,B 0,C 180,E1 -12385.888,E2 -12385.888} C_VEL
LIN {X 0,Y 375.953,Z 337.257,A -85,B 0,C 180,E1 -12389.687,E2 -12389.687} C_VEL
LIN {X 0,Y 375.925,Z 337.276,A -85,B 0,C 180,E1 -12392.136,E2 -12392.136} C_VEL
LIN {X 0,Y 375.962,Z 337.273,A -85,B 0,C 180,E1 -12395.717,E2 -12395.717} C_VEL
LIN {X 0,Y 375.97,Z 337.273,A -85,B 0,C 180,E1 -12399.197,E2 -12399.197} C_VEL
LIN {X 0,Y 376.022,Z 337.267,A -85,B 0,C 180,E1 -12402.6,E2 -12402.6} C_VEL
LIN {X 0,Y 376.079,Z 337.262,A -85,B 0,C 180,E1 -12406.343,E2 -12406.343} C_VEL
LIN {X 0,Y 376.094,Z 337.26,A -85,B 0,C 180,E1 -12410.318,E2 -12410.318} C_VEL
LIN {X 0,Y 376.187,Z 337.244,A -85,B 0,C 180,E1 -12413.564,E2 -12413.564} C_VEL
LIN {X 0,Y 376.326,Z 337.225,A -85,B 0,C 180,E1 -12417.86,E2 -12417.86} C_VEL
LIN {X 0,Y 376.333,Z 337.224,A -85,B 0,C 180,E1 -12422.141,E2 -12422.141} C_VEL
LIN {X 0,Y 376.196,Z 337.244,A -85,B 0,C 180,E1 -12426.569,E2 -12426.569} C_VEL
LIN {X 0,Y 376.102,Z 337.261,A -85,B 0,C 180,E1 -12429.682,E2 -12429.682} C_VEL
LIN {X 0,Y 376.08,Z 337.263,A -85,B 0,C 180,E1 -12433.658,E2 -12433.658} C_VEL
LIN {X 0,Y 376.023,Z 337.269,A -85,B 0,C 180,E1 -12437.401,E2 -12437.401} C_VEL
LIN {X 0,Y 375.971,Z 337.273,A -85,B 0,C 180,E1 -12440.833,E2 -12440.833} C_VEL
LIN {X 0,Y 375.982,Z 337.272,A -85,B 0,C 180,E1 -12444.283,E2 -12444.283} C_VEL
LIN {X 0,Y 376.013,Z 337.275,A -85,B 0,C 180,E1 -12446.653,E2 -12446.653} C_VEL
LIN {X 0,Y 375.958,Z 337.279,A -85,B 0,C 180,E1 -12450.314,E2 -12450.314} C_VEL
LIN {X 0,Y 375.955,Z 337.277,A -85,B 0,C 180,E1 -12454.113,E2 -12454.113} C_VEL
LIN {X 0,Y 375.948,Z 337.277,A -85,B 0,C 180,E1 -12456.742,E2 -12456.742} C_VEL
LIN {X 0,Y 375.983,Z 337.272,A -85,B 0,C 180,E1 -12459.972,E2 -12459.972} C_VEL
LIN {X 0,Y 375.927,Z 337.283,A -85,B 0,C 180,E1 -12463.767,E2 -12463.767} C_VEL
LIN {X 0,Y 375.932,Z 337.282,A -85,B 0,C 180,E1 -12466.812,E2 -12466.812} C_VEL
LIN {X 0,Y 375.963,Z 337.279,A -85,B 0,C 180,E1 -12470.539,E2 -12470.539} C_VEL
LIN {X 0,Y 376.009,Z 337.354,A -85,B 0,C 180,E1 -12474.55,E2 -12474.55} C_VEL
LIN {X 0,Y 378.54,Z 348.14,A -85,B 0,C 180,E1 -12477.476,E2 -12477.476} C_VEL
LIN {X 0,Y 387.447,Z 368.151,A -85,B 0,C 180,E1 -12478.615,E2 -12478.615} C_VEL
LIN {X 0,Y 389.604,Z 377.158,A -85,B 0,C 180,E1 -12478.966,E2 -12478.966} C_VEL
LIN {X 0,Y 387.388,Z 483.062,A -85,B 0,C 180,E1 -12480.969,E2 -12480.969} C_VEL
LIN {X 0,Y 386.745,Z 497.736,A -85,B 0,C 180,E1 -12481.436,E2 -12481.436} C_VEL
LIN {X 0,Y 385.821,Z 511.658,A -85,B 0,C 180,E1 -12482.102,E2 -12482.102} C_VEL
LIN {X 0,Y 384.592,Z 525.278,A -85,B 0,C 180,E1 -12482.979,E2 -12482.979} C_VEL
LIN {X 0,Y 383.218,Z 538.619,A -85,B 0,C 180,E1 -12484.096,E2 -12484.096} C_VEL
LIN {X 0,Y 381.788,Z 549.686,A -85,B 0,C 180,E1 -12485.243,E2 -12485.243} C_VEL
LIN {X 0,Y 380.432,Z 560.369,A -85,B 0,C 180,E1 -12486.598,E2 -12486.598} C_VEL
LIN {X 0,Y 379.136,Z 570.938,A -85,B 0,C 180,E1 -12488.24,E2 -12488.24} C_VEL
LIN {X 0,Y 377.863,Z 579.613,A -85,B 0,C 180,E1 -12489.874,E2 -12489.874} C_VEL
LIN {X 0,Y 376.938,Z 586.79,A -85,B 0,C 180,E1 -12491.521,E2 -12491.521} C_VEL
LIN {X 0,Y 376.131,Z 592.725,A -85,B 0,C 180,E1 -12493.165,E2 -12493.165} C_VEL
LIN {X 0,Y 375.371,Z 599.033,A -85,B 0,C 180,E1 -12495.36,E2 -12495.36} C_VEL
LIN {X 0,Y 374.98,Z 602.732,A -85,B 0,C 180,E1 -12497.062,E2 -12497.062} C_VEL
LIN {X 0,Y 374.601,Z 606.105,A -85,B 0,C 180,E1 -12499.187,E2 -12499.187} C_VEL
LIN {X 0,Y 374.477,Z 608.179,A -85,B 0,C 180,E1 -12501.365,E2 -12501.365} C_VEL
LIN {X 0,Y 374.534,Z 608.905,A -85,B 0,C 180,E1 -12503.536,E2 -12503.536} C_VEL
LIN {X 0,Y 374.53,Z 608.308,A -85,B 0,C 180,E1 -12505.695,E2 -12505.695} C_VEL
LIN {X 0,Y 374.558,Z 606.379,A -85,B 0,C 180,E1 -12507.849,E2 -12507.849} C_VEL
LIN {X 0,Y 374.707,Z 603.071,A -85,B 0,C 180,E1 -12510,E2 -12510} C_VEL
LIN {X 0,Y 374.973,Z 598.304,A -85,B 0,C 180,E1 -12512.148,E2 -12512.148} C_VEL
LIN {X 0,Y 375.557,Z 591.918,A -85,B 0,C 180,E1 -12514.293,E2 -12514.293} C_VEL
LIN {X 0,Y 376.417,Z 584.81,A -85,B 0,C 180,E1 -12516.163,E2 -12516.163} C_VEL
LIN {X 0,Y 377.459,Z 576.039,A -85,B 0,C 180,E1 -12518.027,E2 -12518.027} C_VEL
LIN {X 0,Y 378.343,Z 566.871,A -85,B 0,C 180,E1 -12519.624,E2 -12519.624} C_VEL
LIN {X 0,Y 378.946,Z 561.686,A -85,B 0,C 180,E1 -12520.398,E2 -12520.398} C_VEL
LIN {X 0,Y 378.797,Z 557.414,A -85,B 0,C 180,E1 -12521.013,E2 -12521.013} C_VEL
LIN {X 0,Y 376.888,Z 550.305,A -85,B 0,C 180,E1 -12522.02,E2 -12522.02} C_VEL
LIN {X 0,Y 374.922,Z 542.851,A -85,B 0,C 180,E1 -12522.967,E2 -12522.967} C_VEL
LIN {X 0,Y 374.676,Z 537.976,A -85,B 0,C 180,E1 -12523.48,E2 -12523.48} C_VEL
LIN {X 0,Y 375.765,Z 526.135,A -85,B 0,C 180,E1 -12524.486,E2 -12524.486} C_VEL
LIN {X 0,Y 376.875,Z 512.219,A -85,B 0,C 180,E1 -12525.41,E2 -12525.41} C_VEL
LIN {X 0,Y 377.739,Z 498.119,A -85,B 0,C 180,E1 -12526.101,E2 -12526.101} C_VEL
LIN {X 0,Y 378.301,Z 484.282,A -85,B 0,C 180,E1 -12526.562,E2 -12526.562} C_VEL
LIN {X 0,Y 380.249,Z 377.3,A -85,B 0,C 180,E1 -12528.609,E2 -12528.609} C_VEL
LIN {X 0,Y 377.599,Z 364.865,A -85,B 0,C 180,E1 -12529.028,E2 -12529.028} C_VEL
LIN {X 0,Y 371.046,Z 347.798,A -85,B 0,C 180,E1 -12529.84,E2 -12529.84} C_VEL
LIN {X 0,Y 368.928,Z 338.156,A -85,B 0,C 180,E1 -12532.395,E2 -12532.395} C_VEL
LIN {X 0,Y 369.002,Z 338.148,A -85,B 0,C 180,E1 -12535.979,E2 -12535.979} C_VEL
LIN {X 0,Y 368.916,Z 338.155,A -85,B 0,C 180,E1 -12539.689,E2 -12539.689} C_VEL
LIN {X 0,Y 368.897,Z 338.157,A -85,B 0,C 180,E1 -12543.042,E2 -12543.042} C_VEL
LIN {X 0,Y 368.918,Z 338.151,A -85,B 0,C 180,E1 -12546.196,E2 -12546.196} C_VEL
LIN {X 0,Y 368.904,Z 338.156,A -85,B 0,C 180,E1 -12548.952,E2 -12548.952} C_VEL
LIN {X 0,Y 368.88,Z 338.159,A -85,B 0,C 180,E1 -12552.008,E2 -12552.008} C_VEL
LIN {X 0,Y 368.877,Z 338.158,A -85,B 0,C 180,E1 -12555.175,E2 -12555.175} C_VEL
LIN {X 0,Y 368.878,Z 338.154,A -85,B 0,C 180,E1 -12558.176,E2 -12558.176} C_VEL
LIN {X 0,Y 368.902,Z 338.155,A -85,B 0,C 180,E1 -12561.359,E2 -12561.359} C_VEL
LIN {X 0,Y 368.931,Z 338.156,A -85,B 0,C 180,E1 -12565.145,E2 -12565.145} C_VEL
LIN {X 0,Y 368.923,Z 338.157,A -85,B 0,C 180,E1 -12569.045,E2 -12569.045} C_VEL
LIN {X 0,Y 368.955,Z 338.14,A -85,B 0,C 180,E1 -12571.561,E2 -12571.561} C_VEL
LIN {X 0,Y 368.937,Z 338.156,A -85,B 0,C 180,E1 -12575.223,E2 -12575.223} C_VEL
LIN {X 0,Y 368.912,Z 338.143,A -85,B 0,C 180,E1 -12578.98,E2 -12578.98} C_VEL
LIN {X 0,Y 368.982,Z 338.143,A -85,B 0,C 180,E1 -12582.256,E2 -12582.256} C_VEL
LIN {X 0,Y 369.028,Z 338.133,A -85,B 0,C 180,E1 -12586.227,E2 -12586.227} C_VEL
LIN {X 0,Y 369.052,Z 338.134,A -85,B 0,C 180,E1 -12590.131,E2 -12590.131} C_VEL
LIN {X 0,Y 369.168,Z 338.116,A -85,B 0,C 180,E1 -12593.441,E2 -12593.441} C_VEL
LIN {X 0,Y 369.294,Z 338.102,A -85,B 0,C 180,E1 -12597.818,E2 -12597.818} C_VEL
LIN {X 0,Y 369.282,Z 338.104,A -85,B 0,C 180,E1 -12602.181,E2 -12602.181} C_VEL
LIN {X 0,Y 369.143,Z 338.129,A -85,B 0,C 180,E1 -12606.559,E2 -12606.559} C_VEL
LIN {X 0,Y 369.049,Z 338.128,A -85,B 0,C 180,E1 -12609.868,E2 -12609.868} C_VEL
LIN {X 0,Y 369.027,Z 338.141,A -85,B 0,C 180,E1 -12613.772,E2 -12613.772} C_VEL
LIN {X 0,Y 368.981,Z 338.145,A -85,B 0,C 180,E1 -12617.743,E2 -12617.743} C_VEL
LIN {X 0,Y 368.9,Z 338.145,A -85,B 0,C 180,E1 -12621.221,E2 -12621.221} C_VEL
LIN {X 0,Y 368.923,Z 338.149,A -85,B 0,C 180,E1 -12624.778,E2 -12624.778} C_VEL
LIN {X 0,Y 368.907,Z 338.155,A -85,B 0,C 180,E1 -12628.442,E2 -12628.442} C_VEL
LIN {X 0,Y 368.889,Z 338.16,A -85,B 0,C 180,E1 -12632.239,E2 -12632.239} C_VEL
LIN {X 0,Y 368.921,Z 338.152,A -85,B 0,C 180,E1 -12635.002,E2 -12635.002} C_VEL
LIN {X 0,Y 368.901,Z 338.156,A -85,B 0,C 180,E1 -12638.641,E2 -12638.641} C_VEL
LIN {X 0,Y 368.874,Z 338.152,A -85,B 0,C 180,E1 -12642.01,E2 -12642.01} C_VEL
LIN {X 0,Y 368.874,Z 338.16,A -85,B 0,C 180,E1 -12645.176,E2 -12645.176} C_VEL
LIN {X 0,Y 368.877,Z 338.161,A -85,B 0,C 180,E1 -12648.178,E2 -12648.178} C_VEL
LIN {X 0,Y 368.902,Z 338.163,A -85,B 0,C 180,E1 -12651.361,E2 -12651.361} C_VEL
LIN {X 0,Y 368.933,Z 338.159,A -85,B 0,C 180,E1 -12655.147,E2 -12655.147} C_VEL
LIN {X 0,Y 368.935,Z 338.319,A -85,B 0,C 180,E1 -12657.985,E2 -12657.985} C_VEL
LIN {X 0,Y 372.112,Z 351.959,A -85,B 0,C 180,E1 -12661.21,E2 -12661.21} C_VEL
LIN {X 0,Y 374.014,Z 362.11,A -85,B 0,C 180,E1 -12663.496,E2 -12663.496} C_VEL
LIN {X 0,Y 373.601,Z 366.663,A -85,B 0,C 180,E1 -12664.387,E2 -12664.387} C_VEL
LIN {X 0,Y 379.737,Z 402.04,A -85,B 0,C 180,E1 -12665.494,E2 -12665.494} C_VEL
LIN {X 0,Y 379.041,Z 450.14,A -85,B 0,C 180,E1 -12666.413,E2 -12666.413} C_VEL
LIN {X 0,Y 377.93,Z 505.288,A -85,B 0,C 180,E1 -12667.483,E2 -12667.483} C_VEL
LIN {X 0,Y 377.243,Z 518.968,A -85,B 0,C 180,E1 -12667.945,E2 -12667.945} C_VEL
LIN {X 0,Y 376.348,Z 531.924,A -85,B 0,C 180,E1 -12668.574,E2 -12668.574} C_VEL
LIN {X 0,Y 375.233,Z 545.604,A -85,B 0,C 180,E1 -12669.469,E2 -12669.469} C_VEL
LIN {X 0,Y 374.026,Z 558.102,A -85,B 0,C 180,E1 -12670.518,E2 -12670.518} C_VEL
LIN {X 0,Y 372.7,Z 569.776,A -85,B 0,C 180,E1 -12671.73,E2 -12671.73} C_VEL
LIN {X 0,Y 371.402,Z 581.463,A -85,B 0,C 180,E1 -12673.228,E2 -12673.228} C_VEL
LIN {X 0,Y 370.249,Z 591.906,A -85,B 0,C 180,E1 -12674.871,E2 -12674.871} C_VEL
LIN {X 0,Y 369.423,Z 600.658,A -85,B 0,C 180,E1 -12676.553,E2 -12676.553} C_VEL
LIN {X 0,Y 368.576,Z 608.737,A -85,B 0,C 180,E1 -12678.451,E2 -12678.451} C_VEL
LIN {X 0,Y 368.023,Z 614.513,A -85,B 0,C 180,E1 -12680.104,E2 -12680.104} C_VEL
LIN {X 0,Y 367.705,Z 619.211,A -85,B 0,C 180,E1 -12681.759,E2 -12681.759} C_VEL
LIN {X 0,Y 367.515,Z 624.017,A -85,B 0,C 180,E1 -12683.932,E2 -12683.932} C_VEL
LIN {X 0,Y 367.445,Z 626.703,A -85,B 0,C 180,E1 -12685.612,E2 -12685.612} C_VEL
LIN {X 0,Y 367.371,Z 628.984,A -85,B 0,C 180,E1 -12687.807,E2 -12687.807} C_VEL
LIN {X 0,Y 367.455,Z 629.911,A -85,B 0,C 180,E1 -12690,E2 -12690} C_VEL
LIN {X 0,Y 367.356,Z 629.497,A -85,B 0,C 180,E1 -12692.193,E2 -12692.193} C_VEL
LIN {X 0,Y 367.42,Z 627.753,A -85,B 0,C 180,E1 -12694.388,E2 -12694.388} C_VEL
LIN {X 0,Y 367.561,Z 624.64,A -85,B 0,C 180,E1 -12696.588,E2 -12696.588} C_VEL
LIN {X 0,Y 367.861,Z 620.069,A -85,B 0,C 180,E1 -12698.791,E2 -12698.791} C_VEL
LIN {X 0,Y 368.419,Z 613.857,A -85,B 0,C 180,E1 -12700.997,E2 -12700.997} C_VEL
LIN {X 0,Y 369.389,Z 606.954,A -85,B 0,C 180,E1 -12702.918,E2 -12702.918} C_VEL
LIN {X 0,Y 370.411,Z 598.412,A -85,B 0,C 180,E1 -12704.84,E2 -12704.84} C_VEL
LIN {X 0,Y 371.659,Z 589.507,A -85,B 0,C 180,E1 -12706.478,E2 -12706.478} C_VEL
LIN {X 0,Y 372.881,Z 580.695,A -85,B 0,C 180,E1 -12707.835,E2 -12707.835} C_VEL
LIN {X 0,Y 374.569,Z 569.037,A -85,B 0,C 180,E1 -12709.31,E2 -12709.31} C_VEL
LIN {X 0,Y 376.075,Z 557.392,A -85,B 0,C 180,E1 -12710.511,E2 -12710.511} C_VEL
LIN {X 0,Y 377.521,Z 544.331,A -85,B 0,C 180,E1 -12711.593,E2 -12711.593} C_VEL
LIN {X 0,Y 378.728,Z 531.306,A -85,B 0,C 180,E1 -12712.431,E2 -12712.431} C_VEL
LIN {X 0,Y 379.907,Z 516.776,A -85,B 0,C 180,E1 -12713.111,E2 -12713.111} C_VEL
LIN {X 0,Y 380.673,Z 503.439,A -85,B 0,C 180,E1 -12713.53,E2 -12713.53} C_VEL
LIN {X 0,Y 382.787,Z 403.276,A -85,B 0,C 180,E1 -12715.461,E2 -12715.461} C_VEL
LIN {X 0,Y 377.786,Z 377.44,A -85,B 0,C 180,E1 -12716.402,E2 -12716.402} C_VEL
LIN {X 0,Y 375.251,Z 366.056,A -85,B 0,C 180,E1 -12716.889,E2 -12716.889} C_VEL
LIN {X 0,Y 373.963,Z 358.617,A -85,B 0,C 180,E1 -12718.634,E2 -12718.634} C_VEL
LIN {X 0,Y 371.136,Z 346.869,A -85,B 0,C 180,E1 -12721.555,E2 -12721.555} C_VEL
LIN {X 0,Y 368.931,Z 338.156,A -85,B 0,C 180,E1 -12723.861,E2 -12723.861} C_VEL
LIN {X 0,Y 368.899,Z 338.146,A -85,B 0,C 180,E1 -12727.562,E2 -12727.562} C_VEL
LIN {X 0,Y 368.905,Z 338.143,A -85,B 0,C 180,E1 -12730.37,E2 -12730.37} C_VEL
LIN {X 0,Y 368.876,Z 338.154,A -85,B 0,C 180,E1 -12733.615,E2 -12733.615} C_VEL
LIN {X 0,Y 368.879,Z 338.157,A -85,B 0,C 180,E1 -12736.695,E2 -12736.695} C_VEL
LIN {X 0,Y 368.905,Z 338.155,A -85,B 0,C 180,E1 -12739.642,E2 -12739.642} C_VEL
LIN {X 0,Y 368.894,Z 338.157,A -85,B 0,C 180,E1 -12743.144,E2 -12743.144} C_VEL
LIN {X 0,Y 368.888,Z 338.16,A -85,B 0,C 180,E1 -12746.461,E2 -12746.461} C_VEL
LIN {X 0,Y 368.904,Z 338.141,A -85,B 0,C 180,E1 -12749.044,E2 -12749.044} C_VEL
LIN {X 0,Y 368.907,Z 338.143,A -85,B 0,C 180,E1 -12751.558,E2 -12751.558} C_VEL
LIN {X 0,Y 368.916,Z 338.151,A -85,B 0,C 180,E1 -12755.222,E2 -12755.222} C_VEL
LIN {X 0,Y 368.91,Z 338.152,A -85,B 0,C 180,E1 -12758.98,E2 -12758.98} C_VEL
LIN {X 0,Y 368.981,Z 338.146,A -85,B 0,C 180,E1 -12762.257,E2 -12762.257} C_VEL
LIN {X 0,Y 369.027,Z 338.141,A -85,B 0,C 180,E1 -12766.228,E2 -12766.228} C_VEL
LIN {X 0,Y 369.045,Z 338.14,A -85,B 0,C 180,E1 -12770.131,E2 -12770.131} C_VEL
LIN {X 0,Y 369.148,Z 338.12,A -85,B 0,C 180,E1 -12773.441,E2 -12773.441} C_VEL
LIN {X 0,Y 369.29,Z 338.101,A -85,B 0,C 180,E1 -12777.819,E2 -12777.819} C_VEL
LIN {X 0,Y 369.297,Z 338.1,A -85,B 0,C 180,E1 -12782.182,E2 -12782.182} C_VEL
LIN {X 0,Y 369.168,Z 338.121,A -85,B 0,C 180,E1 -12786.559,E2 -12786.559} C_VEL
LIN {X 0,Y 369.052,Z 338.138,A -85,B 0,C 180,E1 -12789.869,E2 -12789.869} C_VEL
LIN {X 0,Y 369.028,Z 338.141,A -85,B 0,C 180,E1 -12793.773,E2 -12793.773} C_VEL
LIN {X 0,Y 368.983,Z 338.146,A -85,B 0,C 180,E1 -12797.744,E2 -12797.744} C_VEL
LIN {X 0,Y 368.902,Z 338.155,A -85,B 0,C 180,E1 -12801.222,E2 -12801.222} C_VEL
LIN {X 0,Y 368.948,Z 338.148,A -85,B 0,C 180,E1 -12804.777,E2 -12804.777} C_VEL
LIN {X 0,Y 368.956,Z 338.148,A -85,B 0,C 180,E1 -12807.205,E2 -12807.205} C_VEL
LIN {X 0,Y 368.924,Z 338.151,A -85,B 0,C 180,E1 -12810.955,E2 -12810.955} C_VEL
LIN {X 0,Y 368.924,Z 338.153,A -85,B 0,C 180,E1 -12815.002,E2 -12815.002} C_VEL
LIN {X 0,Y 368.903,Z 338.159,A -85,B 0,C 180,E1 -12818.641,E2 -12818.641} C_VEL
LIN {X 0,Y 368.878,Z 338.161,A -85,B 0,C 180,E1 -12822.011,E2 -12822.011} C_VEL
LIN {X 0,Y 368.877,Z 338.161,A -85,B 0,C 180,E1 -12825.177,E2 -12825.177} C_VEL
LIN {X 0,Y 368.881,Z 338.163,A -85,B 0,C 180,E1 -12828.179,E2 -12828.179} C_VEL
LIN {X 0,Y 368.91,Z 338.158,A -85,B 0,C 180,E1 -12831.36,E2 -12831.36} C_VEL
LIN {X 0,Y 368.956,Z 338.172,A -85,B 0,C 180,E1 -12834.03,E2 -12834.03} C_VEL
LIN {X 0,Y 371.41,Z 348.332,A -85,B 0,C 180,E1 -12836.868,E2 -12836.868} C_VEL
LIN {X 0,Y 381.116,Z 369.956,A -85,B 0,C 180,E1 -12838.15,E2 -12838.15} C_VEL
LIN {X 0,Y 382.548,Z 374.825,A -85,B 0,C 180,E1 -12838.367,E2 -12838.367} C_VEL
LIN {X 0,Y 383.295,Z 378.321,A -85,B 0,C 180,E1 -12838.499,E2 -12838.499} C_VEL
LIN {X 0,Y 380.911,Z 484.497,A -85,B 0,C 180,E1 -12840.541,E2 -12840.541} C_VEL
LIN {X 0,Y 380.276,Z 498.613,A -85,B 0,C 180,E1 -12841.017,E2 -12841.017} C_VEL
LIN {X 0,Y 379.358,Z 511.782,A -85,B 0,C 180,E1 -12841.659,E2 -12841.659} C_VEL
LIN {X 0,Y 378.179,Z 524.341,A -85,B 0,C 180,E1 -12842.467,E2 -12842.467} C_VEL
LIN {X 0,Y 376.917,Z 536.901,A -85,B 0,C 180,E1 -12843.511,E2 -12843.511} C_VEL
LIN {X 0,Y 375.195,Z 549.247,A -85,B 0,C 180,E1 -12844.778,E2 -12844.778} C_VEL
LIN {X 0,Y 373.767,Z 560.037,A -85,B 0,C 180,E1 -12846.155,E2 -12846.155} C_VEL
LIN {X 0,Y 372.41,Z 570.696,A -85,B 0,C 180,E1 -12847.826,E2 -12847.826} C_VEL
LIN {X 0,Y 371.072,Z 579.445,A -85,B 0,C 180,E1 -12849.49,E2 -12849.49} C_VEL
LIN {X 0,Y 369.912,Z 587.757,A -85,B 0,C 180,E1 -12851.434,E2 -12851.434} C_VEL
LIN {X 0,Y 368.973,Z 594.459,A -85,B 0,C 180,E1 -12853.399,E2 -12853.399} C_VEL
LIN {X 0,Y 368.233,Z 600.342,A -85,B 0,C 180,E1 -12855.634,E2 -12855.634} C_VEL
LIN {X 0,Y 367.732,Z 604.624,A -85,B 0,C 180,E1 -12857.865,E2 -12857.865} C_VEL
LIN {X 0,Y 367.397,Z 607.44,A -85,B 0,C 180,E1 -12860.087,E2 -12860.087} C_VEL
LIN {X 0,Y 367.398,Z 608.878,A -85,B 0,C 180,E1 -12862.305,E2 -12862.305} C_VEL
LIN {X 0,Y 367.43,Z 608.985,A -85,B 0,C 180,E1 -12864.512,E2 -12864.512} C_VEL
LIN {X 0,Y 367.402,Z 607.777,A -85,B 0,C 180,E1 -12866.71,E2 -12866.71} C_VEL
LIN {X 0,Y 367.572,Z 605.22,A -85,B 0,C 180,E1 -12868.904,E2 -12868.904} C_VEL
LIN {X 0,Y 367.745,Z 601.247,A -85,B 0,C 180,E1 -12871.095,E2 -12871.095} C_VEL
LIN {X 0,Y 368.176,Z 595.742,A -85,B 0,C 180,E1 -12873.283,E2 -12873.283} C_VEL
LIN {X 0,Y 368.832,Z 589.529,A -85,B 0,C 180,E1 -12875.193,E2 -12875.193} C_VEL
LIN {X 0,Y 369.809,Z 581.796,A -85,B 0,C 180,E1 -12877.096,E2 -12877.096} C_VEL
LIN {X 0,Y 370.809,Z 573.73,A -85,B 0,C 180,E1 -12878.721,E2 -12878.721} C_VEL
LIN {X 0,Y 371.628,Z 565.575,A -85,B 0,C 180,E1 -12880.11,E2 -12880.11} C_VEL
LIN {X 0,Y 372.869,Z 554.544,A -85,B 0,C 180,E1 -12881.662,E2 -12881.662} C_VEL
LIN {X 0,Y 374.209,Z 542.611,A -85,B 0,C 180,E1 -12883.024,E2 -12883.024} C_VEL
LIN {X 0,Y 374.676,Z 537.976,A -85,B 0,C 180,E1 -12883.48,E2 -12883.48} C_VEL
LIN {X 0,Y 374.435,Z 533.027,A -85,B 0,C 180,E1 -12883.967,E2 -12883.967} C_VEL
LIN {X 0,Y 372.475,Z 524.804,A -85,B 0,C 180,E1 -12884.77,E2 -12884.77} C_VEL
LIN {X 0,Y 370.566,Z 516.335,A -85,B 0,C 180,E1 -12885.499,E2 -12885.499} C_VEL
LIN {X 0,Y 370.304,Z 510.93,A -85,B 0,C 180,E1 -12885.859,E2 -12885.859} C_VEL
LIN {X 0,Y 371.209,Z 496.748,A -85,B 0,C 180,E1 -12886.533,E2 -12886.533} C_VEL
LIN {X 0,Y 371.694,Z 483.261,A -85,B 0,C 180,E1 -12886.971,E2 -12886.971} C_VEL
LIN {X 0,Y 373.657,Z 378.3,A -85,B 0,C 180,E1 -12889.009,E2 -12889.009} C_VEL
LIN {X 0,Y 371.326,Z 367.392,A -85,B 0,C 180,E1 -12889.387,E2 -12889.387} C_VEL
LIN {X 0,Y 364.547,Z 349.998,A -85,B 0,C 180,E1 -12890.215,E2 -12890.215} C_VEL
LIN {X 0,Y 363.835,Z 347.965,A -85,B 0,C 180,E1 -12890.346,E2 -12890.346} C_VEL
LIN {X 0,Y 361.881,Z 339.032,A -85,B 0,C 180,E1 -12892.78,E2 -12892.78} C_VEL
LIN {X 0,Y 361.956,Z 339.024,A -85,B 0,C 180,E1 -12896.524,E2 -12896.524} C_VEL
LIN {X 0,Y 361.874,Z 339.033,A -85,B 0,C 180,E1 -12900.327,E2 -12900.327} C_VEL
LIN {X 0,Y 361.855,Z 339.033,A -85,B 0,C 180,E1 -12904.279,E2 -12904.279} C_VEL
LIN {X 0,Y 361.871,Z 339.032,A -85,B 0,C 180,E1 -12907.223,E2 -12907.223} C_VEL
LIN {X 0,Y 361.834,Z 339.021,A -85,B 0,C 180,E1 -12910.754,E2 -12910.754} C_VEL
LIN {X 0,Y 361.814,Z 339.036,A -85,B 0,C 180,E1 -12914.367,E2 -12914.367} C_VEL
LIN {X 0,Y 361.832,Z 339.035,A -85,B 0,C 180,E1 -12917.567,E2 -12917.567} C_VEL
LIN {X 0,Y 361.864,Z 339.035,A -85,B 0,C 180,E1 -12920.972,E2 -12920.972} C_VEL
LIN {X 0,Y 361.869,Z 339.033,A -85,B 0,C 180,E1 -12924.654,E2 -12924.654} C_VEL
LIN {X 0,Y 361.831,Z 339.035,A -85,B 0,C 180,E1 -12928.369,E2 -12928.369} C_VEL
LIN {X 0,Y 361.894,Z 339.026,A -85,B 0,C 180,E1 -12930.954,E2 -12930.954} C_VEL
LIN {X 0,Y 361.902,Z 339.026,A -85,B 0,C 180,E1 -12934.707,E2 -12934.707} C_VEL
LIN {X 0,Y 361.846,Z 339.03,A -85,B 0,C 180,E1 -12938.344,E2 -12938.344} C_VEL
LIN {X 0,Y 361.912,Z 339.023,A -85,B 0,C 180,E1 -12942.084,E2 -12942.084} C_VEL
LIN {X 0,Y 361.952,Z 339.015,A -85,B 0,C 180,E1 -12945.379,E2 -12945.379} C_VEL
LIN {X 0,Y 361.958,Z 339.012,A -85,B 0,C 180,E1 -12948.804,E2 -12948.804} C_VEL
LIN {X 0,Y 362.084,Z 339.006,A -85,B 0,C 180,E1 -12952.191,E2 -12952.191} C_VEL
LIN {X 0,Y 362.091,Z 338.993,A -85,B 0,C 180,E1 -12954.43,E2 -12954.43} C_VEL
LIN {X 0,Y 362.257,Z 338.978,A -85,B 0,C 180,E1 -12957.776,E2 -12957.776} C_VEL
LIN {X 0,Y 362.244,Z 338.98,A -85,B 0,C 180,E1 -12962.223,E2 -12962.223} C_VEL
LIN {X 0,Y 362.107,Z 339.004,A -85,B 0,C 180,E1 -12966.687,E2 -12966.687} C_VEL
LIN {X 0,Y 361.986,Z 339.008,A -85,B 0,C 180,E1 -12970.063,E2 -12970.063} C_VEL
LIN {X 0,Y 361.988,Z 339.019,A -85,B 0,C 180,E1 -12973.899,E2 -12973.899} C_VEL
LIN {X 0,Y 361.917,Z 339.023,A -85,B 0,C 180,E1 -12976.934,E2 -12976.934} C_VEL
LIN {X 0,Y 361.873,Z 339.023,A -85,B 0,C 180,E1 -12980.461,E2 -12980.461} C_VEL
LIN {X 0,Y 361.884,Z 339.032,A -85,B 0,C 180,E1 -12984.113,E2 -12984.113} C_VEL
LIN {X 0,Y 361.838,Z 339.035,A -85,B 0,C 180,E1 -12987.785,E2 -12987.785} C_VEL
LIN {X 0,Y 361.838,Z 339.032,A -85,B 0,C 180,E1 -12991.286,E2 -12991.286} C_VEL
LIN {X 0,Y 361.846,Z 339.034,A -85,B 0,C 180,E1 -12994.281,E2 -12994.281} C_VEL
LIN {X 0,Y 361.856,Z 339.033,A -85,B 0,C 180,E1 -12997.224,E2 -12997.224} C_VEL
LIN {X 0,Y 361.828,Z 339.03,A -85,B 0,C 180,E1 -13000.756,E2 -13000.756} C_VEL
LIN {X 0,Y 361.811,Z 339.039,A -85,B 0,C 180,E1 -13004.369,E2 -13004.369} C_VEL
LIN {X 0,Y 361.83,Z 339.041,A -85,B 0,C 180,E1 -13007.569,E2 -13007.569} C_VEL
LIN {X 0,Y 361.863,Z 339.038,A -85,B 0,C 180,E1 -13010.974,E2 -13010.974} C_VEL
LIN {X 0,Y 361.87,Z 339.038,A -85,B 0,C 180,E1 -13014.656,E2 -13014.656} C_VEL
LIN {X 0,Y 361.874,Z 339.043,A -85,B 0,C 180,E1 -13017.555,E2 -13017.555} C_VEL
LIN {X 0,Y 365.141,Z 353.127,A -85,B 0,C 180,E1 -13020.964,E2 -13020.964} C_VEL
LIN {X 0,Y 367.075,Z 363.094,A -85,B 0,C 180,E1 -13023.262,E2 -13023.262} C_VEL
LIN {X 0,Y 366.844,Z 366.214,A -85,B 0,C 180,E1 -13023.915,E2 -13023.915} C_VEL
LIN {X 0,Y 371.387,Z 392.499,A -85,B 0,C 180,E1 -13024.773,E2 -13024.773} C_VEL
LIN {X 0,Y 373.313,Z 404.784,A -85,B 0,C 180,E1 -13025.148,E2 -13025.148} C_VEL
LIN {X 0,Y 371.376,Z 503.604,A -85,B 0,C 180,E1 -13027.064,E2 -13027.064} C_VEL
LIN {X 0,Y 370.63,Z 517.826,A -85,B 0,C 180,E1 -13027.53,E2 -13027.53} C_VEL
LIN {X 0,Y 369.625,Z 532.168,A -85,B 0,C 180,E1 -13028.238,E2 -13028.238} C_VEL
LIN {X 0,Y 368.481,Z 545.53,A -85,B 0,C 180,E1 -13029.13,E2 -13029.13} C_VEL
LIN {X 0,Y 367.149,Z 558.904,A -85,B 0,C 180,E1 -13030.283,E2 -13030.283} C_VEL
LIN {X 0,Y 365.665,Z 571.587,A -85,B 0,C 180,E1 -13031.656,E2 -13031.656} C_VEL
LIN {X 0,Y 364.318,Z 582.873,A -85,B 0,C 180,E1 -13033.181,E2 -13033.181} C_VEL
LIN {X 0,Y 363.148,Z 592.989,A -85,B 0,C 180,E1 -13034.855,E2 -13034.855} C_VEL
LIN {X 0,Y 362.328,Z 601.388,A -85,B 0,C 180,E1 -13036.541,E2 -13036.541} C_VEL
LIN {X 0,Y 361.444,Z 609.401,A -85,B 0,C 180,E1 -13038.504,E2 -13038.504} C_VEL
LIN {X 0,Y 360.847,Z 615.844,A -85,B 0,C 180,E1 -13040.471,E2 -13040.471} C_VEL
LIN {X 0,Y 360.524,Z 621.548,A -85,B 0,C 180,E1 -13042.721,E2 -13042.721} C_VEL
LIN {X 0,Y 360.381,Z 624.767,A -85,B 0,C 180,E1 -13044.405,E2 -13044.405} C_VEL
LIN {X 0,Y 360.295,Z 627.772,A -85,B 0,C 180,E1 -13046.645,E2 -13046.645} C_VEL
LIN {X 0,Y 360.318,Z 629.396,A -85,B 0,C 180,E1 -13048.882,E2 -13048.882} C_VEL
LIN {X 0,Y 360.358,Z 629.704,A -85,B 0,C 180,E1 -13050,E2 -13050} C_VEL
LIN {X 0,Y 360.26,Z 629.313,A -85,B 0,C 180,E1 -13052.236,E2 -13052.236} C_VEL
LIN {X 0,Y 360.332,Z 627.592,A -85,B 0,C 180,E1 -13054.474,E2 -13054.474} C_VEL
LIN {X 0,Y 360.495,Z 624.503,A -85,B 0,C 180,E1 -13056.717,E2 -13056.717} C_VEL
LIN {X 0,Y 360.809,Z 619.963,A -85,B 0,C 180,E1 -13058.965,E2 -13058.965} C_VEL
LIN {X 0,Y 361.233,Z 615.476,A -85,B 0,C 180,E1 -13060.651,E2 -13060.651} C_VEL
LIN {X 0,Y 362.134,Z 609.028,A -85,B 0,C 180,E1 -13062.611,E2 -13062.611} C_VEL
LIN {X 0,Y 363.126,Z 600.914,A -85,B 0,C 180,E1 -13064.601,E2 -13064.601} C_VEL
LIN {X 0,Y 364.342,Z 592.7,A -85,B 0,C 180,E1 -13066.242,E2 -13066.242} C_VEL
LIN {X 0,Y 365.821,Z 582.681,A -85,B 0,C 180,E1 -13067.901,E2 -13067.901} C_VEL
LIN {X 0,Y 367.545,Z 571.53,A -85,B 0,C 180,E1 -13069.404,E2 -13069.404} C_VEL
LIN {X 0,Y 369.236,Z 559.048,A -85,B 0,C 180,E1 -13070.763,E2 -13070.763} C_VEL
LIN {X 0,Y 370.727,Z 546.642,A -85,B 0,C 180,E1 -13071.845,E2 -13071.845} C_VEL
LIN {X 0,Y 372.042,Z 532.926,A -85,B 0,C 180,E1 -13072.783,E2 -13072.783} C_VEL
LIN {X 0,Y 373.315,Z 519.106,A -85,B 0,C 180,E1 -13073.47,E2 -13073.47} C_VEL
LIN {X 0,Y 374.223,Z 504.758,A -85,B 0,C 180,E1 -13073.961,E2 -13073.961} C_VEL
LIN {X 0,Y 376.186,Z 419.726,A -85,B 0,C 180,E1 -13075.636,E2 -13075.636} C_VEL
LIN {X 0,Y 376.442,Z 403.951,A -85,B 0,C 180,E1 -13075.95,E2 -13075.95} C_VEL
LIN {X 0,Y 371.195,Z 377.213,A -85,B 0,C 180,E1 -13076.96,E2 -13076.96} C_VEL
LIN {X 0,Y 368.878,Z 367.932,A -85,B 0,C 180,E1 -13077.363,E2 -13077.363} C_VEL
LIN {X 0,Y 368.228,Z 365.945,A -85,B 0,C 180,E1 -13077.474,E2 -13077.474} C_VEL
LIN {X 0,Y 365.898,Z 354.897,A -85,B 0,C 180,E1 -13080.193,E2 -13080.193} C_VEL
LIN {X 0,Y 362.45,Z 341.274,A -85,B 0,C 180,E1 -13083.77,E2 -13083.77} C_VEL
LIN {X 0,Y 361.897,Z 339.032,A -85,B 0,C 180,E1 -13084.443,E2 -13084.443} C_VEL
LIN {X 0,Y 361.864,Z 339.029,A -85,B 0,C 180,E1 -13088.424,E2 -13088.424} C_VEL
LIN {X 0,Y 361.822,Z 339.03,A -85,B 0,C 180,E1 -13091.33,E2 -13091.33} C_VEL
LIN {X 0,Y 361.812,Z 339.037,A -85,B 0,C 180,E1 -13094.368,E2 -13094.368} C_VEL
LIN {X 0,Y 361.83,Z 339.033,A -85,B 0,C 180,E1 -13097.567,E2 -13097.567} C_VEL
